(* Logix 5000 project; controller Tekno_ASRS vendor 1 type 14 code 147 rev 20.11; software revision 20.01 *)
// ASRS control program for Tekno ASRS

TASK MainTask (continuous, watchdog 500 ms) : MainProgram
TASK SafetyTask (periodic, rate 160 ms, priority 10, watchdog 20 ms) : SafetyProgram

MODULES
   Local : vendor 1 type 14 code 147 (ICP 0, rev 20.11)
      IOComms : vendor 1 type 12 code 200 (ICP 2, Ethernet 192.168.10.207, rev 5.1, Input RPI 500 ms)
         SpatulaYAxis : vendor 1 type 123 code 50 (Ethernet 192.168.10.202, rev 5.1, Output RPI 20 ms)
             : vendor 1 type 123 code 8192 (DPI 5, rev 4.1)
         XAxis : vendor 1 type 37 code 23 (Ethernet 192.168.10.200, rev 5.1, MotionDiagnostics RPI 1 ms, MotionSync RPI 6 ms)
         ZAxis : vendor 1 type 37 code 23 (Ethernet 192.168.10.201, rev 5.1, MotionDiagnostics RPI 1 ms, MotionSync RPI 6 ms)
         StationaryIO : 1734-AENT (Ethernet 192.168.10.204, rev 3.7, Output RPI 80 ms)
            StationaryIn1 : 1734-IB8 (PointIO 1, rev 3.1)
            StationaryIn3 : 1734-IB8 (PointIO 3, rev 3.1)
            StationaryIn2 : 1734-IB8 (PointIO 2, rev 3.1)
            StationaryIn4 : 1734-IB8 (PointIO 4, rev 3.1)
            StationaryStrainIn1 : vendor 1 type 0 code 20 (PointIO 5, rev 1.1, Output RPI 80 ms)
            StationarOut8 : 1734-OB8 (PointIO 8, rev 3.1)
            StationarySafetyIn1 : vendor 1 type 35 code 15 (PointIO 7, rev 1.1, Input RPI 40 ms)
            StationarySafetyOut1 : vendor 1 type 35 code 16 (PointIO 6, rev 1.1, Input RPI 320 ms, Output RPI 160 ms)
         ShuttleIO : 1734-AENT (Ethernet 192.168.10.203, rev 3.1, Output RPI 20 ms)
            ShuttleIn2 : 1734-IB8 (PointIO 2, rev 3.1)
            ShuttleIn1 : 1734-IB8 (PointIO 1, rev 3.1)
            ShuttleStrainIn1 : vendor 1 type 0 code 20 (PointIO 3, rev 1.1, Output RPI 80 ms)
            ShuttleStrainIn2 : vendor 1 type 0 code 20 (PointIO 4, rev 1.1, Output RPI 80 ms)
            ShuttleOut2 : 1734-OB8 (PointIO 10, rev 3.1)
            ShuttleOut1 : 1734-OB8 (PointIO 5, rev 3.1)
            ShuttleSafetyIn1 : vendor 1 type 35 code 15 (PointIO 7, rev 1.1, Input RPI 40 ms, Output RPI 160 ms)
            ShuttleSafetyIn2 : vendor 1 type 35 code 15 (PointIO 9, rev 1.1, Input RPI 40 ms, Output RPI 160 ms)
            ShuttleSafetyOut1 : vendor 1 type 35 code 16 (PointIO 6, rev 1.1, Input RPI 40 ms, Output RPI 160 ms)
            ShuttleSafetyOut2 : vendor 1 type 35 code 16 (PointIO 8, rev 1.1, Input RPI 40 ms, Output RPI 160 ms)
      @b5ff5b04@:Partner : vendor 1 type 14 code 146 (ICP 1, rev 20.11)   // ASRS control program for Tekno ASRS
END_MODULES

TYPE ASRS_Status :
STRUCT
   RtRowObstruction : DINT;
   LfRowObstruction : DINT;
END_STRUCT
END_TYPE

TYPE BayPos :
STRUCT
   AAxis : DINT;
   BAxis : DINT;
END_STRUCT
END_TYPE

TYPE Configuration :
STRUCT
   MaxASpeed : REAL;
   MinASpeed : REAL;
   MaxAAcc : REAL;
   MaxADec : REAL;
   AAccelJerk : REAL;
   ADecelJerk : REAL;
   MaxBSpeed : REAL;
   MinBSpeed : REAL;
   MaxBAcc : REAL;
   MaxBDec : REAL;
   BAccelJerk : REAL;
   BDecelJerk : REAL;
   SpatulaOffset : DINT;
   JogADirection : DINT;
   JogBDirection : DINT;
   AllowABSynch : BOOL;
END_STRUCT
END_TYPE

TYPE HMI_Commands :
STRUCT
   CfgEndAAxis : DINT;
   CfgEndBAxis : DINT;
   CfgStrtAAxis : DINT;
   CfgStrtBAxis : DINT;
   MaxA : DINT;
   MaxB : DINT;
   MaxC : DINT;
   GoToALocation : DINT;
   GoToBLocation : DINT;
   XLftStrainScaleSet : DINT;
   XRtStrainScaleSet : DINT;
   ZForeRtStrainScaleSet : DINT;
   ZForeLftStrainScaleSet : DINT;
   ZAftRtStrainScaleSet : DINT;
   ZAftLftStrainScaleSet : DINT;
   AGridLoc : DINT;
   BGridLoc : DINT;
   CGridLoc : DINT;
   XStrainLeftMvV : REAL;
   XStrainRightMvV : REAL;
   ZAftStrainLeftMvV : REAL;
   ZAftStrainRightMvV : REAL;
   ZForeStrainLeftMvV : REAL;
   ZForeStrainRightMvV : REAL;
   HMIStart : BOOL;
   HMIStop : BOOL;
   HMIReset : BOOL;
   JogAAxisEn : BOOL;
   JogAFwd : BOOL;
   JogARev : BOOL;
   JogBAxisEn : BOOL;
   JogBFwd : BOOL;
   JogBRev : BOOL;
   JogCAxisEn : BOOL;
   JogCFwd : BOOL;
   JogCRev : BOOL;
   ManMode : BOOL;
   ZAftRtClrTare : BOOL;
   ZAftRtTare : BOOL;
   ZAftLtClrTare : BOOL;
   ZAftLtTare : BOOL;
   ZForRTClrTare : BOOL;
   ZForRtTare : BOOL;
   ZForLtClrTare : BOOL;
   ZForLtTare : BOOL;
   XLtClrTare : BOOL;
   XLtTare : BOOL;
   XRtClrTare : BOOL;
   XRtTare : BOOL;
   SUIndPos : BOOL;
   XStCalMode : BOOL;
   XStRunMode : BOOL;
   ZAftStCalMode : BOOL;
   ZAftStRunMode : BOOL;
   ZForStCalMode : BOOL;
   ZForStRunMode : BOOL;
   GoToBay : BOOL;
   GoToHome : BOOL;
   MatrixSetUp : BOOL;
   ClearCurrent : BOOL;
   ClearQueue : BOOL;
   DemoStart : BOOL;
   DemoStop : BOOL;
   SpatulaHome : BOOL;
END_STRUCT
END_TYPE

TYPE HMI_Data :
STRUCT
   Status : HMI_Status;
   Faults : HMI_Faults;
END_STRUCT
END_TYPE

TYPE HMI_Faults :
STRUCT
   AAxisFault : DINT;
   BAxisFault : DINT;
   SystemFault : BOOL;
   AftAreaScanner : BOOL;
   EstopSafetyGate : BOOL;
   ForeAreaScanner : BOOL;
   PalmButtons : BOOL;
   RowObstruction : BOOL;
   XTension : BOOL;
   ZAftLeft : BOOL;
   ZAftRight : BOOL;
   ZForeLeft : BOOL;
   ZForeRight : BOOL;
   ShuttleFault : BOOL;
   XAxisMtrSideEOT : BOOL;
   XAxisPnlSideEOT : BOOL;
   ZAxisUpEOT : BOOL;
   ZAxisDnEOT : BOOL;
   ZLatchFault : BOOL;
   AGVLghtCurFlt : BOOL;
END_STRUCT
END_TYPE

TYPE HMI_Status :
STRUCT
   CurrentAPos : REAL;
   CurrentBPos : REAL;
   CurrentCPos : REAL;
   XStrainLeftWeight : DINT;
   XStrainRightWeight : DINT;
   ZAftStrainLeftWeight : DINT;
   ZAftStrainRightWeight : DINT;
   ZForeStrainLeftWeight : DINT;
   ZForeStrainRightWeight : DINT;
   QueuedTasks : DINT;
   AAxisStatus : DINT;
   BAxisStatus : DINT;
   CurrentTaskCommand : SINT;
   CurrentTaskBayAPos : SINT;
   CurrentTaskBayBPos : SINT;
   CurrentTaskBayCPos : SINT;
   CurrentTaskParameter1 : SINT;
   CurrentTaskParameter2 : SINT;
   Auto : BOOL;
   ManOnBoard : BOOL;
   AreaWarning : BOOL;
   ManGateClosed : BOOL;
   BackGateInstalled : BOOL;
   DrivesOn : BOOL;
   SpatulaHome : BOOL;
   SystemRunning : BOOL;
   ZLAftLft : BOOL;
   ZLAftRgt : BOOL;
   ZLForeLft : BOOL;
   ZLForeRgt : BOOL;
   FrontAreaWarn : BOOL;
   RearAreaWarn : BOOL;
   Footswitch : BOOL;
   XAxisBrk : BOOL;
   ZAxisBrk : BOOL;
   PalmButtonLeft : BOOL;
   PalmButtonright : BOOL;
END_STRUCT
END_TYPE

TYPE Messaging :
STRUCT
   Command : SINT;
   CoordinateA : SINT;
   CoordinateB : SINT;
   CoordinateC : SINT;
   Parameter1 : SINT;
   Parameter2 : SINT;
   Sequence : DINT;
END_STRUCT
END_TYPE

TYPE Position :
STRUCT
   Apos : REAL;
   Bpos : REAL;
   Cpos : REAL[10];
END_STRUCT
END_TYPE

TYPE Strain :
STRUCT
   LeftScaleSet : DINT;
   LeftAutoCalSet : DINT;
   LeftWeight : DINT;
   LeftRaw : DINT;
   LeftCal : DINT;
   RightScaleSet : DINT;
   RightAutoCalSet : DINT;
   RightWeight : DINT;
   RightRaw : DINT;
   RightCal : DINT;
   CfgAveSampCnt : DINT;
   LeftMvV : REAL;
   RightMvV : REAL;
   LeftEnAutoCal : BOOL;
   RightEnAutoCal : BOOL;
END_STRUCT
END_TYPE

TYPE Task :
STRUCT
   Command : SINT;
   BayAPos : SINT;
   BayBPos : SINT;
   BayCPos : SINT;
   Parameter1 : SINT;
   Parameter2 : SINT;
END_STRUCT
END_TYPE

VAR_GLOBAL   (* controller tags *)
   A : DINT;
   AAxis : AXIS_CIP_DRIVE;
   AAxisJog : MOTION_INSTRUCTION := (FLAGS := 33554432);
   AAxisMAM : MOTION_INSTRUCTION := (FLAGS := 167772160, PC := 1);
   AAxisMove : BOOL := 1;
   AAxisOn : MOTION_INSTRUCTION := (FLAGS := 536870912, DN := 1, STATE := 1);
   AAXisReset : MOTION_INSTRUCTION := (FLAGS := 536870912, DN := 1, STATE := 1);
   AAxisSODelay : TIMER := (PRE := 200);
   AAxisState : DINT;
   AAxisStop : MOTION_INSTRUCTION := (FLAGS := 33554432);
   ABayPos : DINT;
   ABGrid : Position[100,20] := ([0,0].Apos := 475.0, [0,0].Bpos := 0.02327277, [0,1].Apos := 63.589, [0,1].Bpos := 6.6, [0,1].Cpos[1] := -196128.0, [0,2].Apos := 677.48, [0,2].Bpos := 6.6, [0,2].Cpos[1] := -196128.0, [0,3].Apos := 46.1, [0,3].Bpos := 77.4, [0,3].Cpos[1] := -196128.0, [0,4].Apos := 80.1, [0,4].Bpos := 77.4, [0,4].Cpos[1] := -196128.0, [0,5].Apos := 660.18, [0,5].Bpos := 77.4, [0,5].Cpos[1] := -196128.0, [0,6].Apos := 694.375, [0,6].Bpos := 77.4, [0,6].Cpos[1] := -196128.0, [0,7].Apos := 415.0, [0,8].Apos := 415.0, [0,9].Apos := 415.0, [0,10].Apos := 415.0, [0,11].Apos := 415.0, [0,12].Apos := 415.0, [0,13].Apos := 415.0, [0,14].Apos := 415.0, [0,15].Apos := 415.0, [0,16].Apos := 415.0, [0,17].Apos := 415.0, [0,18].Apos := 415.0, [0,19].Apos := 415.0, [1,0].Apos := 415.0, [1,1].Apos := -42.35, [1,2].Apos := -42.35, [1,2].Bpos := 7.87817, [1,3].Apos := -42.35, [1,3].Bpos := 39.87817, [1,4].Apos := -42.35, [1,4].Bpos := 71.878174, [1,5].Apos := -42.35, [1,5].Bpos := 103.878174, [1,6].Apos := -42.35, [1,6].Bpos := 135.87817, [1,7].Apos := -42.35, [1,7].Bpos := 167.87817, [1,8].Apos := -42.35, [1,8].Bpos := 199.87817, [1,9].Apos := -42.35, [1,9].Bpos := 215.0, [1,10].Apos := 415.0, [1,11].Apos := 415.0, [1,12].Apos := 415.0, [1,13].Apos := 415.0, [1,14].Apos := 415.0, [1,15].Apos := 415.0, [1,16].Apos := 415.0, [1,17].Apos := 415.0, [1,18].Apos := 415.0,
        [1,19].Apos := 415.0, [2,0].Apos := 415.0, [2,1].Apos := -42.35, [2,2].Apos := -42.35, [2,2].Bpos := 7.87817, [2,3].Apos := -42.35, [2,3].Bpos := 39.87817, [2,4].Apos := -42.35, [2,4].Bpos := 71.878174, [2,5].Apos := -42.35, [2,5].Bpos := 103.878174, [2,6].Apos := -42.35, [2,6].Bpos := 135.87817, [2,7].Apos := -42.35, [2,7].Bpos := 167.87817, [2,8].Apos := -42.35, [2,8].Bpos := 199.87817, [2,9].Apos := -42.35, [2,9].Bpos := 215.0, [2,10].Apos := 415.0, [2,11].Apos := 415.0, [2,12].Apos := 415.0, [2,13].Apos := 415.0, [2,14].Apos := 415.0, [2,15].Apos := 415.0, [2,16].Apos := 415.0, [2,17].Apos := 415.0, [2,18].Apos := 415.0, [2,19].Apos := 415.0, [3,0].Apos := 415.0, [3,1].Apos := -26.905, [3,2].Apos := -26.905, [3,2].Bpos := 7.87817, [3,3].Apos := -26.905, [3,3].Bpos := 39.87817, [3,4].Apos := -26.905, [3,4].Bpos := 71.878174, [3,5].Apos := -26.905, [3,5].Bpos := 103.878174, [3,6].Apos := -26.905, [3,6].Bpos := 135.87817, [3,7].Apos := -26.905, [3,7].Bpos := 167.87817, [3,8].Apos := -26.905, [3,8].Bpos := 199.87817, [3,9].Apos := -26.905, [3,9].Bpos := 215.0, [3,10].Apos := 415.0, [3,11].Apos := 415.0, [3,12].Apos := 415.0, [3,13].Apos := 415.0, [3,14].Apos := 415.0, [3,15].Apos := 415.0, [3,16].Apos := 415.0, [3,17].Apos := 415.0, [3,18].Apos := 415.0, [3,19].Apos := 415.0, [4,0].Apos := 415.0, [4,1].Apos := -1.235, [4,2].Apos := -1.235,
        [4,2].Bpos := 7.87817, [4,3].Apos := -1.235, [4,3].Bpos := 39.87817, [4,4].Apos := -1.235, [4,4].Bpos := 71.878174, [4,5].Apos := -1.235, [4,5].Bpos := 103.878174, [4,6].Apos := -1.235, [4,6].Bpos := 135.87817, [4,7].Apos := -1.235, [4,7].Bpos := 167.87817, [4,8].Apos := -1.235, [4,8].Bpos := 199.87817, [4,9].Apos := -1.235, [4,9].Bpos := 215.0, [4,10].Apos := 415.0, [4,11].Apos := 415.0, [4,12].Apos := 415.0, [4,13].Apos := 415.0, [4,14].Apos := 415.0, [4,15].Apos := 415.0, [4,16].Apos := 415.0, [4,17].Apos := 415.0, [4,18].Apos := 415.0, [4,19].Apos := 415.0, [5,0].Apos := 415.0, [5,1].Apos := 24.435026, [5,2].Apos := 24.435026, [5,2].Bpos := 7.87817, [5,3].Apos := 24.435026, [5,3].Bpos := 39.87817, [5,4].Apos := 24.435026, [5,4].Bpos := 71.878174, [5,5].Apos := 24.435026, [5,5].Bpos := 103.878174, [5,6].Apos := 24.435026, [5,6].Bpos := 135.87817, [5,7].Apos := 24.435026, [5,7].Bpos := 167.87817, [5,8].Apos := 24.435026, [5,8].Bpos := 199.87817, [5,9].Apos := 24.435026, [5,9].Bpos := 215.0, [5,10].Apos := 415.0, [5,11].Apos := 415.0, [5,12].Apos := 415.0, [5,13].Apos := 415.0, [5,14].Apos := 415.0, [5,15].Apos := 415.0, [5,16].Apos := 415.0, [5,17].Apos := 415.0, [5,18].Apos := 415.0, [5,19].Apos := 415.0, [6,0].Apos := 415.0, [6,1].Apos := 50.105618, [6,2].Apos := 50.105618, [6,2].Bpos := 7.87817, [6,3].Apos := 50.105618, [6,3].Bpos := 39.87817, [6,4].Apos := 50.105618,
        [6,4].Bpos := 71.878174, [6,5].Apos := 50.105618, [6,5].Bpos := 103.878174, [6,6].Apos := 50.105618, [6,6].Bpos := 135.87817, [6,7].Apos := 50.105618, [6,7].Bpos := 167.87817, [6,8].Apos := 50.105618, [6,8].Bpos := 199.87817, [6,9].Apos := 50.105618, [6,9].Bpos := 215.0, [6,10].Apos := 415.0, [6,11].Apos := 415.0, [6,12].Apos := 415.0, [6,13].Apos := 415.0, [6,14].Apos := 415.0, [6,15].Apos := 415.0, [6,16].Apos := 415.0, [6,17].Apos := 415.0, [6,18].Apos := 415.0, [6,19].Apos := 415.0, [7,0].Apos := 415.0, [7,1].Apos := 75.77621, [7,2].Apos := 75.77621, [7,2].Bpos := 7.87817, [7,3].Apos := 75.77621, [7,3].Bpos := 39.87817, [7,4].Apos := 75.77621, [7,4].Bpos := 71.878174, [7,5].Apos := 75.77621, [7,5].Bpos := 103.878174, [7,6].Apos := 75.77621, [7,6].Bpos := 135.87817, [7,7].Apos := 75.77621, [7,7].Bpos := 167.87817, [7,8].Apos := 75.77621, [7,8].Bpos := 199.87817, [7,9].Apos := 75.77621, [7,9].Bpos := 215.0, [7,10].Apos := 415.0, [7,11].Apos := 415.0, [7,12].Apos := 415.0, [7,13].Apos := 415.0, [7,14].Apos := 415.0, [7,15].Apos := 415.0, [7,16].Apos := 415.0, [7,17].Apos := 415.0, [7,18].Apos := 415.0, [7,19].Apos := 415.0, [8,0].Apos := 415.0, [8,1].Apos := 101.4468, [8,2].Apos := 101.4468, [8,2].Bpos := 7.87817, [8,3].Apos := 101.4468, [8,3].Bpos := 39.87817, [8,4].Apos := 101.4468, [8,4].Bpos := 71.878174, [8,5].Apos := 101.4468, [8,5].Bpos := 103.878174, [8,6].Apos := 101.4468,
        [8,6].Bpos := 135.87817, [8,7].Apos := 101.4468, [8,7].Bpos := 167.87817, [8,8].Apos := 101.4468, [8,8].Bpos := 199.87817, [8,9].Apos := 101.4468, [8,9].Bpos := 215.0, [8,10].Apos := 415.0, [8,11].Apos := 415.0, [8,12].Apos := 415.0, [8,13].Apos := 415.0, [8,14].Apos := 415.0, [8,15].Apos := 415.0, [8,16].Apos := 415.0, [8,17].Apos := 415.0, [8,18].Apos := 415.0, [8,19].Apos := 415.0, [9,0].Apos := 415.0, [9,1].Apos := 127.11739, [9,2].Apos := 127.11739, [9,2].Bpos := 7.87817, [9,3].Apos := 127.11739, [9,3].Bpos := 39.87817, [9,4].Apos := 127.11739, [9,4].Bpos := 71.878174, [9,5].Apos := 127.11739, [9,5].Bpos := 103.878174, [9,6].Apos := 127.11739, [9,6].Bpos := 135.87817, [9,7].Apos := 127.11739, [9,7].Bpos := 167.87817, [9,8].Apos := 127.11739, [9,8].Bpos := 199.87817, [9,9].Apos := 127.11739, [9,9].Bpos := 215.0, [9,10].Apos := 415.0, [9,11].Apos := 415.0, [9,12].Apos := 415.0, [9,13].Apos := 415.0, [9,14].Apos := 415.0, [9,15].Apos := 415.0, [9,16].Apos := 415.0, [9,17].Apos := 415.0, [9,18].Apos := 415.0, [9,19].Apos := 415.0, [10,0].Apos := 415.0, [10,1].Apos := 152.78798, [10,2].Apos := 152.78798, [10,2].Bpos := 7.87817, [10,3].Apos := 152.78798, [10,3].Bpos := 39.87817, [10,4].Apos := 152.78798, [10,4].Bpos := 71.878174, [10,5].Apos := 152.78798, [10,5].Bpos := 103.878174, [10,6].Apos := 152.78798, [10,6].Bpos := 135.87817, [10,7].Apos := 152.78798, [10,7].Bpos := 167.87817, [10,8].Apos := 152.78798,
        [10,8].Bpos := 199.87817, [10,9].Apos := 152.78798, [10,9].Bpos := 215.0, [10,10].Apos := 415.0, [10,11].Apos := 415.0, [10,12].Apos := 415.0, [10,13].Apos := 415.0, [10,14].Apos := 415.0, [10,15].Apos := 415.0, [10,16].Apos := 415.0, [10,17].Apos := 415.0, [10,18].Apos := 415.0, [10,19].Apos := 415.0, [11,0].Apos := 415.0, [11,1].Apos := 178.45857, [11,2].Apos := 178.45857, [11,2].Bpos := 7.87817, [11,3].Apos := 178.45857, [11,3].Bpos := 39.87817, [11,4].Apos := 178.45857, [11,4].Bpos := 71.878174, [11,5].Apos := 178.45857, [11,5].Bpos := 103.878174, [11,6].Apos := 178.45857, [11,6].Bpos := 135.87817, [11,7].Apos := 178.45857, [11,7].Bpos := 167.87817, [11,8].Apos := 178.45857, [11,8].Bpos := 199.87817, [11,9].Apos := 178.45857, [11,9].Bpos := 215.0, [11,10].Apos := 415.0, [11,11].Apos := 415.0, [11,12].Apos := 415.0, [11,13].Apos := 415.0, [11,14].Apos := 415.0, [11,15].Apos := 415.0, [11,16].Apos := 415.0, [11,17].Apos := 415.0, [11,18].Apos := 415.0, [11,19].Apos := 415.0, [12,0].Apos := 415.0, [12,1].Apos := 204.12917, [12,2].Apos := 204.12917, [12,2].Bpos := 7.87817, [12,3].Apos := 204.12917, [12,3].Bpos := 39.87817, [12,4].Apos := 204.12917, [12,4].Bpos := 71.878174, [12,5].Apos := 204.12917, [12,5].Bpos := 103.878174, [12,6].Apos := 204.12917, [12,6].Bpos := 135.87817, [12,7].Apos := 204.12917, [12,7].Bpos := 167.87817, [12,8].Apos := 204.12917, [12,8].Bpos := 199.87817, [12,9].Apos := 204.12917, [12,9].Bpos := 215.0, [12,10].Apos := 415.0,
        [12,11].Apos := 415.0, [12,12].Apos := 415.0, [12,13].Apos := 415.0, [12,14].Apos := 415.0, [12,15].Apos := 415.0, [12,16].Apos := 415.0, [12,17].Apos := 415.0, [12,18].Apos := 415.0, [12,19].Apos := 415.0, [13,0].Apos := 415.0, [13,1].Apos := 229.79976, [13,2].Apos := 229.79976, [13,2].Bpos := 7.87817, [13,3].Apos := 229.79976, [13,3].Bpos := 39.87817, [13,4].Apos := 229.79976, [13,4].Bpos := 71.878174, [13,5].Apos := 229.79976, [13,5].Bpos := 103.878174, [13,6].Apos := 229.79976, [13,6].Bpos := 135.87817, [13,7].Apos := 229.79976, [13,7].Bpos := 167.87817, [13,8].Apos := 229.79976, [13,8].Bpos := 199.87817, [13,9].Apos := 229.79976, [13,9].Bpos := 215.0, [13,10].Apos := 415.0, [13,11].Apos := 415.0, [13,12].Apos := 415.0, [13,13].Apos := 415.0, [13,14].Apos := 415.0, [13,15].Apos := 415.0, [13,16].Apos := 415.0, [13,17].Apos := 415.0, [13,18].Apos := 415.0, [13,19].Apos := 415.0, [14,0].Apos := 415.0, [14,1].Apos := 255.47035, [14,2].Apos := 255.47035, [14,2].Bpos := 7.87817, [14,3].Apos := 255.47035, [14,3].Bpos := 39.87817, [14,4].Apos := 255.47035, [14,4].Bpos := 71.878174, [14,5].Apos := 255.47035, [14,5].Bpos := 103.878174, [14,6].Apos := 255.47035, [14,6].Bpos := 135.87817, [14,7].Apos := 255.47035, [14,7].Bpos := 167.87817, [14,8].Apos := 255.47035, [14,8].Bpos := 199.87817, [14,9].Apos := 255.47035, [14,9].Bpos := 215.0, [14,10].Apos := 415.0, [14,11].Apos := 415.0, [14,12].Apos := 415.0, [14,13].Apos := 415.0, [14,14].Apos := 415.0,
        [14,15].Apos := 415.0, [14,16].Apos := 415.0, [14,17].Apos := 415.0, [14,18].Apos := 415.0, [14,19].Apos := 415.0, [15,0].Apos := 415.0, [15,1].Apos := 281.14093, [15,2].Apos := 281.14093, [15,2].Bpos := 7.87817, [15,3].Apos := 281.14093, [15,3].Bpos := 39.87817, [15,4].Apos := 281.14093, [15,4].Bpos := 71.878174, [15,5].Apos := 281.14093, [15,5].Bpos := 103.878174, [15,6].Apos := 281.14093, [15,6].Bpos := 135.87817, [15,7].Apos := 281.14093, [15,7].Bpos := 167.87817, [15,8].Apos := 281.14093, [15,8].Bpos := 199.87817, [15,9].Apos := 281.14093, [15,9].Bpos := 215.0, [15,10].Apos := 415.0, [15,11].Apos := 415.0, [15,12].Apos := 415.0, [15,13].Apos := 415.0, [15,14].Apos := 415.0, [15,15].Apos := 415.0, [15,16].Apos := 415.0, [15,17].Apos := 415.0, [15,18].Apos := 415.0, [15,19].Apos := 415.0, [16,0].Apos := 415.0, [16,1].Apos := 306.81152, [16,2].Apos := 306.81152, [16,2].Bpos := 7.87817, [16,3].Apos := 306.81152, [16,3].Bpos := 39.87817, [16,4].Apos := 306.81152, [16,4].Bpos := 71.878174, [16,5].Apos := 306.81152, [16,5].Bpos := 103.878174, [16,6].Apos := 306.81152, [16,6].Bpos := 135.87817, [16,7].Apos := 306.81152, [16,7].Bpos := 167.87817, [16,8].Apos := 306.81152, [16,8].Bpos := 199.87817, [16,9].Apos := 306.81152, [16,9].Bpos := 215.0, [16,10].Apos := 415.0, [16,11].Apos := 415.0, [16,12].Apos := 415.0, [16,13].Apos := 415.0, [16,14].Apos := 415.0, [16,15].Apos := 415.0, [16,16].Apos := 415.0, [16,17].Apos := 415.0, [16,18].Apos := 415.0,
        [16,19].Apos := 415.0, [17,0].Apos := 415.0, [17,1].Apos := 332.48212, [17,2].Apos := 332.48212, [17,2].Bpos := 7.87817, [17,3].Apos := 332.48212, [17,3].Bpos := 39.87817, [17,4].Apos := 332.48212, [17,4].Bpos := 71.878174, [17,5].Apos := 332.48212, [17,5].Bpos := 103.878174, [17,6].Apos := 332.48212, [17,6].Bpos := 135.87817, [17,7].Apos := 332.48212, [17,7].Bpos := 167.87817, [17,8].Apos := 332.48212, [17,8].Bpos := 199.87817, [17,9].Apos := 332.48212, [17,9].Bpos := 215.0, [17,10].Apos := 415.0, [17,11].Apos := 415.0, [17,12].Apos := 415.0, [17,13].Apos := 415.0, [17,14].Apos := 415.0, [17,15].Apos := 415.0, [17,16].Apos := 415.0, [17,17].Apos := 415.0, [17,18].Apos := 415.0, [17,19].Apos := 415.0, [18,0].Apos := 415.0, [18,1].Apos := 358.1527, [18,2].Apos := 358.1527, [18,2].Bpos := 7.87817, [18,3].Apos := 358.1527, [18,3].Bpos := 39.87817, [18,4].Apos := 358.1527, [18,4].Bpos := 71.878174, [18,5].Apos := 358.1527, [18,5].Bpos := 103.878174, [18,6].Apos := 358.1527, [18,6].Bpos := 135.87817, [18,7].Apos := 358.1527, [18,7].Bpos := 167.87817, [18,8].Apos := 358.1527, [18,8].Bpos := 199.87817, [18,9].Apos := 358.1527, [18,9].Bpos := 215.0, [18,10].Apos := 415.0, [18,11].Apos := 415.0, [18,12].Apos := 415.0, [18,13].Apos := 415.0, [18,14].Apos := 415.0, [18,15].Apos := 415.0, [18,16].Apos := 415.0, [18,17].Apos := 415.0, [18,18].Apos := 415.0, [18,19].Apos := 415.0, [19,0].Apos := 415.0, [19,1].Apos := 383.8233, [19,2].Apos := 383.8233,
        [19,2].Bpos := 7.87817, [19,3].Apos := 383.8233, [19,3].Bpos := 39.87817, [19,4].Apos := 383.8233, [19,4].Bpos := 71.878174, [19,5].Apos := 383.8233, [19,5].Bpos := 103.878174, [19,6].Apos := 383.8233, [19,6].Bpos := 135.87817, [19,7].Apos := 383.8233, [19,7].Bpos := 167.87817, [19,8].Apos := 383.8233, [19,8].Bpos := 199.87817, [19,9].Apos := 383.8233, [19,9].Bpos := 215.0, [19,10].Apos := 415.0, [19,11].Apos := 415.0, [19,12].Apos := 415.0, [19,13].Apos := 415.0, [19,14].Apos := 415.0, [19,15].Apos := 415.0, [19,16].Apos := 415.0, [19,17].Apos := 415.0, [19,18].Apos := 415.0, [19,19].Apos := 415.0, [20,0].Apos := 415.0, [20,1].Apos := 409.4939, [20,2].Apos := 409.4939, [20,2].Bpos := 7.87817, [20,3].Apos := 409.4939, [20,3].Bpos := 39.87817, [20,4].Apos := 409.4939, [20,4].Bpos := 71.878174, [20,5].Apos := 409.4939, [20,5].Bpos := 103.878174, [20,6].Apos := 409.4939, [20,6].Bpos := 135.87817, [20,7].Apos := 409.4939, [20,7].Bpos := 167.87817, [20,8].Apos := 409.4939, [20,8].Bpos := 199.87817, [20,9].Apos := 409.4939, [20,9].Bpos := 215.0, [20,10].Apos := 415.0, [20,11].Apos := 415.0, [20,12].Apos := 415.0, [20,13].Apos := 415.0, [20,14].Apos := 415.0, [20,15].Apos := 415.0, [20,16].Apos := 415.0, [20,17].Apos := 415.0, [20,18].Apos := 415.0, [20,19].Apos := 415.0, [21,0].Apos := 415.0, [21,1].Apos := 435.1645, [21,2].Apos := 435.1645, [21,2].Bpos := 7.87817, [21,3].Apos := 435.1645, [21,3].Bpos := 39.87817, [21,4].Apos := 435.1645,
        [21,4].Bpos := 71.878174, [21,5].Apos := 435.1645, [21,5].Bpos := 103.878174, [21,6].Apos := 435.1645, [21,6].Bpos := 135.87817, [21,7].Apos := 435.1645, [21,7].Bpos := 167.87817, [21,8].Apos := 435.1645, [21,8].Bpos := 199.87817, [21,9].Apos := 435.1645, [21,9].Bpos := 215.0, [21,10].Apos := 415.0, [21,11].Apos := 415.0, [21,12].Apos := 415.0, [21,13].Apos := 415.0, [21,14].Apos := 415.0, [21,15].Apos := 415.0, [21,16].Apos := 415.0, [21,17].Apos := 415.0, [21,18].Apos := 415.0, [21,19].Apos := 415.0, [22,0].Apos := 415.0, [22,1].Apos := 460.83508, [22,2].Apos := 460.83508, [22,2].Bpos := 7.87817, [22,3].Apos := 460.83508, [22,3].Bpos := 39.87817, [22,4].Apos := 460.83508, [22,4].Bpos := 71.878174, [22,5].Apos := 460.83508, [22,5].Bpos := 103.878174, [22,6].Apos := 460.83508, [22,6].Bpos := 135.87817, [22,7].Apos := 460.83508, [22,7].Bpos := 167.87817, [22,8].Apos := 460.83508, [22,8].Bpos := 199.87817, [22,9].Apos := 460.83508, [22,9].Bpos := 215.0, [22,10].Apos := 415.0, [22,11].Apos := 415.0, [22,12].Apos := 415.0, [22,13].Apos := 415.0, [22,14].Apos := 415.0, [22,15].Apos := 415.0, [22,16].Apos := 415.0, [22,17].Apos := 415.0, [22,18].Apos := 415.0, [22,19].Apos := 415.0, [23,0].Apos := 415.0, [23,1].Apos := 486.50568, [23,2].Apos := 486.50568, [23,2].Bpos := 7.87817, [23,3].Apos := 486.50568, [23,3].Bpos := 39.87817, [23,4].Apos := 486.50568, [23,4].Bpos := 71.878174, [23,5].Apos := 486.50568, [23,5].Bpos := 103.878174, [23,6].Apos := 486.50568,
        [23,6].Bpos := 135.87817, [23,7].Apos := 486.50568, [23,7].Bpos := 167.87817, [23,8].Apos := 486.50568, [23,8].Bpos := 199.87817, [23,9].Apos := 486.50568, [23,9].Bpos := 215.0, [23,10].Apos := 415.0, [23,11].Apos := 415.0, [23,12].Apos := 415.0, [23,13].Apos := 415.0, [23,14].Apos := 415.0, [23,15].Apos := 415.0, [23,16].Apos := 415.0, [23,17].Apos := 415.0, [23,18].Apos := 415.0, [23,19].Apos := 415.0, [24,0].Apos := 415.0, [24,1].Apos := 512.1763, [24,2].Apos := 512.1763, [24,2].Bpos := 7.87817, [24,3].Apos := 512.1763, [24,3].Bpos := 39.87817, [24,4].Apos := 512.1763, [24,4].Bpos := 71.878174, [24,5].Apos := 512.1763, [24,5].Bpos := 103.878174, [24,6].Apos := 512.1763, [24,6].Bpos := 135.87817, [24,7].Apos := 512.1763, [24,7].Bpos := 167.87817, [24,8].Apos := 512.1763, [24,8].Bpos := 199.87817, [24,9].Apos := 512.1763, [24,9].Bpos := 215.0, [24,10].Apos := 415.0, [24,11].Apos := 415.0, [24,12].Apos := 415.0, [24,13].Apos := 415.0, [24,14].Apos := 415.0, [24,15].Apos := 415.0, [24,16].Apos := 415.0, [24,17].Apos := 415.0, [24,18].Apos := 415.0, [24,19].Apos := 415.0, [25,0].Apos := 415.0, [25,1].Apos := 537.8468, [25,2].Apos := 537.8468, [25,2].Bpos := 7.87817, [25,3].Apos := 537.8468, [25,3].Bpos := 39.87817, [25,4].Apos := 537.8468, [25,4].Bpos := 71.878174, [25,5].Apos := 537.8468, [25,5].Bpos := 103.878174, [25,6].Apos := 537.8468, [25,6].Bpos := 135.87817, [25,7].Apos := 537.8468, [25,7].Bpos := 167.87817, [25,8].Apos := 537.8468,
        [25,8].Bpos := 199.87817, [25,9].Apos := 537.8468, [25,9].Bpos := 215.0, [25,10].Apos := 415.0, [25,11].Apos := 415.0, [25,12].Apos := 415.0, [25,13].Apos := 415.0, [25,14].Apos := 415.0, [25,15].Apos := 415.0, [25,16].Apos := 415.0, [25,17].Apos := 415.0, [25,18].Apos := 415.0, [25,19].Apos := 415.0, [26,0].Apos := 415.0, [26,1].Apos := 563.5174, [26,2].Apos := 563.5174, [26,2].Bpos := 7.87817, [26,3].Apos := 563.5174, [26,3].Bpos := 39.87817, [26,4].Apos := 563.5174, [26,4].Bpos := 71.878174, [26,5].Apos := 563.5174, [26,5].Bpos := 103.878174, [26,6].Apos := 563.5174, [26,6].Bpos := 135.87817, [26,7].Apos := 563.5174, [26,7].Bpos := 167.87817, [26,8].Apos := 563.5174, [26,8].Bpos := 199.87817, [26,9].Apos := 563.5174, [26,9].Bpos := 215.0, [26,10].Apos := 415.0, [26,11].Apos := 415.0, [26,12].Apos := 415.0, [26,13].Apos := 415.0, [26,14].Apos := 415.0, [26,15].Apos := 415.0, [26,16].Apos := 415.0, [26,17].Apos := 415.0, [26,18].Apos := 415.0, [26,19].Apos := 415.0, [27,0].Apos := 415.0, [27,1].Apos := 589.188, [27,2].Apos := 589.188, [27,2].Bpos := 7.87817, [27,3].Apos := 589.188, [27,3].Bpos := 39.87817, [27,4].Apos := 589.188, [27,4].Bpos := 71.878174, [27,5].Apos := 589.188, [27,5].Bpos := 103.878174, [27,6].Apos := 589.188, [27,6].Bpos := 135.87817, [27,7].Apos := 589.188, [27,7].Bpos := 167.87817, [27,8].Apos := 589.188, [27,8].Bpos := 199.87817, [27,9].Apos := 589.188, [27,9].Bpos := 215.0, [27,10].Apos := 415.0,
        [27,11].Apos := 415.0, [27,12].Apos := 415.0, [27,13].Apos := 415.0, [27,14].Apos := 415.0, [27,15].Apos := 415.0, [27,16].Apos := 415.0, [27,17].Apos := 415.0, [27,18].Apos := 415.0, [27,19].Apos := 415.0, [28,0].Apos := 415.0, [28,1].Apos := 614.8586, [28,2].Apos := 614.8586, [28,2].Bpos := 7.87817, [28,3].Apos := 614.8586, [28,3].Bpos := 39.87817, [28,4].Apos := 614.8586, [28,4].Bpos := 71.878174, [28,5].Apos := 614.8586, [28,5].Bpos := 103.878174, [28,6].Apos := 614.8586, [28,6].Bpos := 135.87817, [28,7].Apos := 614.8586, [28,7].Bpos := 167.87817, [28,8].Apos := 614.8586, [28,8].Bpos := 199.87817, [28,9].Apos := 614.8586, [28,9].Bpos := 215.0, [28,10].Apos := 415.0, [28,11].Apos := 415.0, [28,12].Apos := 415.0, [28,13].Apos := 415.0, [28,14].Apos := 415.0, [28,15].Apos := 415.0, [28,16].Apos := 415.0, [28,17].Apos := 415.0, [28,18].Apos := 415.0, [28,19].Apos := 415.0, [29,0].Apos := 415.0, [29,1].Apos := 640.5292, [29,2].Apos := 640.5292, [29,2].Bpos := 7.87817, [29,3].Apos := 640.5292, [29,3].Bpos := 39.87817, [29,4].Apos := 640.5292, [29,4].Bpos := 71.878174, [29,5].Apos := 640.5292, [29,5].Bpos := 103.878174, [29,6].Apos := 640.5292, [29,6].Bpos := 135.87817, [29,7].Apos := 640.5292, [29,7].Bpos := 167.87817, [29,8].Apos := 640.5292, [29,8].Bpos := 199.87817, [29,9].Apos := 640.5292, [29,9].Bpos := 215.0, [29,10].Apos := 415.0, [29,11].Apos := 415.0, [29,12].Apos := 415.0, [29,13].Apos := 415.0, [29,14].Apos := 415.0,
        [29,15].Apos := 415.0, [29,16].Apos := 415.0, [29,17].Apos := 415.0, [29,18].Apos := 415.0, [29,19].Apos := 415.0, [30,0].Apos := 415.0, [30,1].Apos := 666.19977, [30,2].Apos := 666.19977, [30,2].Bpos := 7.87817, [30,3].Apos := 666.19977, [30,3].Bpos := 39.87817, [30,4].Apos := 666.19977, [30,4].Bpos := 71.878174, [30,5].Apos := 666.19977, [30,5].Bpos := 103.878174, [30,6].Apos := 666.19977, [30,6].Bpos := 135.87817, [30,7].Apos := 666.19977, [30,7].Bpos := 167.87817, [30,8].Apos := 666.19977, [30,8].Bpos := 199.87817, [30,9].Apos := 666.19977, [30,9].Bpos := 215.0, [30,10].Apos := 415.0, [30,11].Apos := 415.0, [30,12].Apos := 415.0, [30,13].Apos := 415.0, [30,14].Apos := 415.0, [30,15].Apos := 415.0, [30,16].Apos := 415.0, [30,17].Apos := 415.0, [30,18].Apos := 415.0, [30,19].Apos := 415.0, [31,0].Apos := 415.0, [31,1].Apos := 691.87036, [31,2].Apos := 691.87036, [31,2].Bpos := 7.87817, [31,3].Apos := 691.87036, [31,3].Bpos := 39.87817, [31,4].Apos := 691.87036, [31,4].Bpos := 71.878174, [31,5].Apos := 691.87036, [31,5].Bpos := 103.878174, [31,6].Apos := 691.87036, [31,6].Bpos := 135.87817, [31,7].Apos := 691.87036, [31,7].Bpos := 167.87817, [31,8].Apos := 691.87036, [31,8].Bpos := 199.87817, [31,9].Apos := 691.87036, [31,9].Bpos := 215.0, [31,10].Apos := 415.0, [31,11].Apos := 415.0, [31,12].Apos := 415.0, [31,13].Apos := 415.0, [31,14].Apos := 415.0, [31,15].Apos := 415.0, [31,16].Apos := 415.0, [31,17].Apos := 415.0, [31,18].Apos := 415.0,
        [31,19].Apos := 415.0, [32,0].Apos := 415.0, [32,1].Apos := 717.54095, [32,2].Apos := 717.54095, [32,2].Bpos := 7.87817, [32,3].Apos := 717.54095, [32,3].Bpos := 39.87817, [32,4].Apos := 717.54095, [32,4].Bpos := 71.878174, [32,5].Apos := 717.54095, [32,5].Bpos := 103.878174, [32,6].Apos := 717.54095, [32,6].Bpos := 135.87817, [32,7].Apos := 717.54095, [32,7].Bpos := 167.87817, [32,8].Apos := 717.54095, [32,8].Bpos := 199.87817, [32,9].Apos := 717.54095, [32,9].Bpos := 215.0, [32,10].Apos := 415.0, [32,11].Apos := 415.0, [32,12].Apos := 415.0, [32,13].Apos := 415.0, [32,14].Apos := 415.0, [32,15].Apos := 415.0, [32,16].Apos := 415.0, [32,17].Apos := 415.0, [32,18].Apos := 415.0, [32,19].Apos := 415.0, [33,0].Apos := 415.0, [33,1].Apos := 743.21155, [33,2].Apos := 743.21155, [33,2].Bpos := 7.87817, [33,3].Apos := 743.21155, [33,3].Bpos := 39.87817, [33,4].Apos := 743.21155, [33,4].Bpos := 71.878174, [33,5].Apos := 743.21155, [33,5].Bpos := 103.878174, [33,6].Apos := 743.21155, [33,6].Bpos := 135.87817, [33,7].Apos := 743.21155, [33,7].Bpos := 167.87817, [33,8].Apos := 743.21155, [33,8].Bpos := 199.87817, [33,9].Apos := 743.21155, [33,9].Bpos := 215.0, [33,10].Apos := 415.0, [33,11].Apos := 415.0, [33,12].Apos := 415.0, [33,13].Apos := 415.0, [33,14].Apos := 415.0, [33,15].Apos := 415.0, [33,16].Apos := 415.0, [33,17].Apos := 415.0, [33,18].Apos := 415.0, [33,19].Apos := 415.0, [34,0].Apos := 415.0, [34,1].Apos := 768.88214, [34,2].Apos := 768.88214,
        [34,2].Bpos := 7.87817, [34,3].Apos := 768.88214, [34,3].Bpos := 39.87817, [34,4].Apos := 768.88214, [34,4].Bpos := 71.878174, [34,5].Apos := 768.88214, [34,5].Bpos := 103.878174, [34,6].Apos := 768.88214, [34,6].Bpos := 135.87817, [34,7].Apos := 768.88214, [34,7].Bpos := 167.87817, [34,8].Apos := 768.88214, [34,8].Bpos := 199.87817, [34,9].Apos := 768.88214, [34,9].Bpos := 215.0, [34,10].Apos := 415.0, [34,11].Apos := 415.0, [34,12].Apos := 415.0, [34,13].Apos := 415.0, [34,14].Apos := 415.0, [34,15].Apos := 415.0, [34,16].Apos := 415.0, [34,17].Apos := 415.0, [34,18].Apos := 415.0, [34,19].Apos := 415.0, [35,0].Apos := 415.0, [35,1].Apos := 794.55273, [35,2].Apos := 794.55273, [35,2].Bpos := 7.87817, [35,3].Apos := 794.55273, [35,3].Bpos := 39.87817, [35,4].Apos := 794.55273, [35,4].Bpos := 71.878174, [35,5].Apos := 794.55273, [35,5].Bpos := 103.878174, [35,6].Apos := 794.55273, [35,6].Bpos := 135.87817, [35,7].Apos := 794.55273, [35,7].Bpos := 167.87817, [35,8].Apos := 794.55273, [35,8].Bpos := 199.87817, [35,9].Apos := 794.55273, [35,9].Bpos := 215.0, [35,10].Apos := 415.0, [35,11].Apos := 415.0, [35,12].Apos := 415.0, [35,13].Apos := 415.0, [35,14].Apos := 415.0, [35,15].Apos := 415.0, [35,16].Apos := 415.0, [35,17].Apos := 415.0, [35,18].Apos := 415.0, [35,19].Apos := 415.0, [36,0].Apos := 415.0, [36,1].Apos := 820.2233, [36,2].Apos := 820.2233, [36,2].Bpos := 7.87817, [36,3].Apos := 820.2233, [36,3].Bpos := 39.87817, [36,4].Apos := 820.2233,
        [36,4].Bpos := 71.878174, [36,5].Apos := 820.2233, [36,5].Bpos := 103.878174, [36,6].Apos := 820.2233, [36,6].Bpos := 135.87817, [36,7].Apos := 820.2233, [36,7].Bpos := 167.87817, [36,8].Apos := 820.2233, [36,8].Bpos := 199.87817, [36,9].Apos := 820.2233, [36,9].Bpos := 215.0, [36,10].Apos := 415.0, [36,11].Apos := 415.0, [36,12].Apos := 415.0, [36,13].Apos := 415.0, [36,14].Apos := 415.0, [36,15].Apos := 415.0, [36,16].Apos := 415.0, [36,17].Apos := 415.0, [36,18].Apos := 415.0, [36,19].Apos := 415.0, [37,0].Apos := 415.0, [37,1].Apos := 845.89, [37,2].Apos := 845.89, [37,2].Bpos := 8.0, [37,3].Apos := 845.89, [37,3].Bpos := 40.0, [37,4].Apos := 845.89, [37,4].Bpos := 72.0, [37,5].Apos := 845.89, [37,5].Bpos := 104.0, [37,6].Apos := 845.89, [37,6].Bpos := 136.0, [37,7].Apos := 845.89, [37,7].Bpos := 168.0, [37,8].Apos := 845.89, [37,8].Bpos := 200.0, [37,9].Apos := 845.89, [37,9].Bpos := 215.0, [37,10].Apos := 415.0, [37,11].Apos := 415.0, [37,12].Apos := 415.0, [37,13].Apos := 415.0, [37,14].Apos := 415.0, [37,15].Apos := 415.0, [37,16].Apos := 415.0, [37,17].Apos := 415.0, [37,18].Apos := 415.0, [37,19].Apos := 415.0, [38,0].Apos := 415.0, [38,1].Apos := 871.6, [38,2].Apos := 871.6, [38,2].Bpos := 8.0, [38,3].Apos := 871.6, [38,3].Bpos := 40.0, [38,4].Apos := 871.6, [38,4].Bpos := 72.0, [38,5].Apos := 871.6, [38,5].Bpos := 104.0, [38,6].Apos := 871.6,
        [38,6].Bpos := 136.0, [38,7].Apos := 871.6, [38,7].Bpos := 168.0, [38,8].Apos := 871.6, [38,8].Bpos := 200.0, [38,9].Apos := 871.6, [38,9].Bpos := 215.0, [38,10].Apos := 415.0, [38,11].Apos := 415.0, [38,12].Apos := 415.0, [38,13].Apos := 415.0, [38,14].Apos := 415.0, [38,15].Apos := 415.0, [38,16].Apos := 415.0, [38,17].Apos := 415.0, [38,18].Apos := 415.0, [38,19].Apos := 415.0, [39,0].Apos := 415.0, [39,1].Apos := 887.0, [39,2].Apos := 887.0, [39,2].Bpos := 8.0, [39,3].Apos := 887.0, [39,3].Bpos := 40.0, [39,4].Apos := 887.0, [39,4].Bpos := 72.0, [39,5].Apos := 887.0, [39,5].Bpos := 104.0, [39,6].Apos := 887.0, [39,6].Bpos := 136.0, [39,7].Apos := 887.0, [39,7].Bpos := 168.0, [39,8].Apos := 887.0, [39,8].Bpos := 200.0, [39,9].Apos := 887.0, [39,9].Bpos := 215.0, [39,10].Apos := 415.0, [39,11].Apos := 415.0, [39,12].Apos := 415.0, [39,13].Apos := 415.0, [39,14].Apos := 415.0, [39,15].Apos := 415.0, [39,16].Apos := 415.0, [39,17].Apos := 415.0, [39,18].Apos := 415.0, [39,19].Apos := 415.0, [40,0].Apos := 415.0, [40,1].Apos := 887.0, [40,2].Apos := 887.0, [40,2].Bpos := 8.0, [40,3].Apos := 887.0, [40,3].Bpos := 40.0, [40,4].Apos := 887.0, [40,4].Bpos := 72.0, [40,5].Apos := 887.0, [40,5].Bpos := 104.0, [40,6].Apos := 887.0, [40,6].Bpos := 136.0, [40,7].Apos := 887.0, [40,7].Bpos := 168.0, [40,8].Apos := 887.0,
        [40,8].Bpos := 200.0, [40,9].Apos := 887.0, [40,9].Bpos := 215.0, [40,10].Apos := 415.0, [40,11].Apos := 415.0, [40,12].Apos := 415.0, [40,13].Apos := 415.0, [40,14].Apos := 415.0, [40,15].Apos := 415.0, [40,16].Apos := 415.0, [40,17].Apos := 415.0, [40,18].Apos := 415.0, [40,19].Apos := 415.0, [41,0].Apos := 415.0, [41,1].Apos := 415.0, [41,2].Apos := 415.0, [41,3].Apos := 415.0, [41,4].Apos := 415.0, [41,5].Apos := 415.0, [41,6].Apos := 415.0, [41,7].Apos := 415.0, [41,8].Apos := 415.0, [41,9].Apos := 415.0, [41,10].Apos := 415.0, [41,11].Apos := 415.0, [41,12].Apos := 415.0, [41,13].Apos := 415.0, [41,14].Apos := 415.0, [41,15].Apos := 415.0, [41,16].Apos := 415.0, [41,17].Apos := 415.0, [41,18].Apos := 415.0, [41,19].Apos := 415.0, [42,0].Apos := 415.0, [42,1].Apos := 415.0, [42,2].Apos := 415.0, [42,3].Apos := 415.0, [42,4].Apos := 415.0, [42,5].Apos := 415.0, [42,6].Apos := 415.0, [42,7].Apos := 415.0, [42,8].Apos := 415.0, [42,9].Apos := 415.0, [42,10].Apos := 415.0, [42,11].Apos := 415.0, [42,12].Apos := 415.0, [42,13].Apos := 415.0, [42,14].Apos := 415.0, [42,15].Apos := 415.0, [42,16].Apos := 415.0, [42,17].Apos := 415.0, [42,18].Apos := 415.0, [42,19].Apos := 415.0, [43,0].Apos := 415.0, [43,1].Apos := 415.0, [43,2].Apos := 415.0, [43,3].Apos := 415.0, [43,4].Apos := 415.0, [43,5].Apos := 415.0, [43,6].Apos := 415.0,
        [43,7].Apos := 415.0, [43,8].Apos := 415.0, [43,9].Apos := 415.0, [43,10].Apos := 415.0, [43,11].Apos := 415.0, [43,12].Apos := 415.0, [43,13].Apos := 415.0, [43,14].Apos := 415.0, [43,15].Apos := 415.0, [43,16].Apos := 415.0, [43,17].Apos := 415.0, [43,18].Apos := 415.0, [43,19].Apos := 415.0, [44,0].Apos := 415.0, [44,1].Apos := 415.0, [44,2].Apos := 415.0, [44,3].Apos := 415.0, [44,4].Apos := 415.0, [44,5].Apos := 415.0, [44,6].Apos := 415.0, [44,7].Apos := 415.0, [44,8].Apos := 415.0, [44,9].Apos := 415.0, [44,10].Apos := 415.0, [44,11].Apos := 415.0, [44,12].Apos := 415.0, [44,13].Apos := 415.0, [44,14].Apos := 415.0, [44,15].Apos := 415.0, [44,16].Apos := 415.0, [44,17].Apos := 415.0, [44,18].Apos := 415.0, [44,19].Apos := 415.0, [45,0].Apos := 415.0, [45,1].Apos := 415.0, [45,2].Apos := 415.0, [45,3].Apos := 415.0, [45,4].Apos := 415.0, [45,5].Apos := 415.0, [45,6].Apos := 415.0, [45,7].Apos := 415.0, [45,8].Apos := 415.0, [45,9].Apos := 415.0, [45,10].Apos := 415.0, [45,11].Apos := 415.0, [45,12].Apos := 415.0, [45,13].Apos := 415.0, [45,14].Apos := 415.0, [45,15].Apos := 415.0, [45,16].Apos := 415.0, [45,17].Apos := 415.0, [45,18].Apos := 415.0, [45,19].Apos := 415.0, [46,0].Apos := 415.0, [46,1].Apos := 415.0, [46,2].Apos := 415.0, [46,3].Apos := 415.0, [46,4].Apos := 415.0, [46,5].Apos := 415.0, [46,6].Apos := 415.0,
        [46,7].Apos := 415.0, [46,8].Apos := 415.0, [46,9].Apos := 415.0, [46,10].Apos := 415.0, [46,11].Apos := 415.0, [46,12].Apos := 415.0, [46,13].Apos := 415.0, [46,14].Apos := 415.0, [46,15].Apos := 415.0, [46,16].Apos := 415.0, [46,17].Apos := 415.0, [46,18].Apos := 415.0, [46,19].Apos := 415.0, [47,0].Apos := 415.0, [47,1].Apos := 415.0, [47,2].Apos := 415.0, [47,3].Apos := 415.0, [47,4].Apos := 415.0, [47,5].Apos := 415.0, [47,6].Apos := 415.0, [47,7].Apos := 415.0, [47,8].Apos := 415.0, [47,9].Apos := 415.0, [47,10].Apos := 415.0, [47,11].Apos := 415.0, [47,12].Apos := 415.0, [47,13].Apos := 415.0, [47,14].Apos := 415.0, [47,15].Apos := 415.0, [47,16].Apos := 415.0, [47,17].Apos := 415.0, [47,18].Apos := 415.0, [47,19].Apos := 415.0, [48,0].Apos := 415.0, [48,1].Apos := 415.0, [48,2].Apos := 415.0, [48,3].Apos := 415.0, [48,4].Apos := 415.0, [48,5].Apos := 415.0, [48,6].Apos := 415.0, [48,7].Apos := 415.0, [48,8].Apos := 415.0, [48,9].Apos := 415.0, [48,10].Apos := 415.0, [48,11].Apos := 415.0, [48,12].Apos := 415.0, [48,13].Apos := 415.0, [48,14].Apos := 415.0, [48,15].Apos := 415.0, [48,16].Apos := 415.0, [48,17].Apos := 415.0, [48,18].Apos := 415.0, [48,19].Apos := 415.0, [49,0].Apos := 415.0, [49,1].Apos := 415.0, [49,2].Apos := 415.0, [49,3].Apos := 415.0, [49,4].Apos := 415.0, [49,5].Apos := 415.0, [49,6].Apos := 415.0,
        [49,7].Apos := 415.0, [49,8].Apos := 415.0, [49,9].Apos := 415.0, [49,10].Apos := 415.0, [49,11].Apos := 415.0, [49,12].Apos := 415.0, [49,13].Apos := 415.0, [49,14].Apos := 415.0, [49,15].Apos := 415.0, [49,16].Apos := 415.0, [49,17].Apos := 415.0, [49,18].Apos := 415.0, [49,19].Apos := 415.0, [50,0].Apos := 415.0, [50,1].Apos := 415.0, [50,2].Apos := 415.0, [50,3].Apos := 415.0, [50,4].Apos := 415.0, [50,5].Apos := 415.0, [50,6].Apos := 415.0, [50,7].Apos := 415.0, [50,8].Apos := 415.0, [50,9].Apos := 415.0, [50,10].Apos := 415.0, [50,11].Apos := 415.0, [50,12].Apos := 415.0, [50,13].Apos := 415.0, [50,14].Apos := 415.0, [50,15].Apos := 415.0, [50,16].Apos := 415.0, [50,17].Apos := 415.0, [50,18].Apos := 415.0, [50,19].Apos := 415.0, [51,0].Apos := 415.0, [51,1].Apos := 415.0, [51,2].Apos := 415.0, [51,3].Apos := 415.0, [51,4].Apos := 415.0, [51,5].Apos := 415.0, [51,6].Apos := 415.0, [51,7].Apos := 415.0, [51,8].Apos := 415.0, [51,9].Apos := 415.0, [51,10].Apos := 415.0, [51,11].Apos := 415.0, [51,12].Apos := 415.0, [51,13].Apos := 415.0, [51,14].Apos := 415.0, [51,15].Apos := 415.0, [51,16].Apos := 415.0, [51,17].Apos := 415.0, [51,18].Apos := 415.0, [51,19].Apos := 415.0, [52,0].Apos := 415.0, [52,1].Apos := 415.0, [52,2].Apos := 415.0, [52,3].Apos := 415.0, [52,4].Apos := 415.0, [52,5].Apos := 415.0, [52,6].Apos := 415.0,
        [52,7].Apos := 415.0, [52,8].Apos := 415.0, [52,9].Apos := 415.0, [52,10].Apos := 415.0, [52,11].Apos := 415.0, [52,12].Apos := 415.0, [52,13].Apos := 415.0, [52,14].Apos := 415.0, [52,15].Apos := 415.0, [52,16].Apos := 415.0, [52,17].Apos := 415.0, [52,18].Apos := 415.0, [52,19].Apos := 415.0, [53,0].Apos := 415.0, [53,1].Apos := 415.0, [53,2].Apos := 415.0, [53,3].Apos := 415.0, [53,4].Apos := 415.0, [53,5].Apos := 415.0, [53,6].Apos := 415.0, [53,7].Apos := 415.0, [53,8].Apos := 415.0, [53,9].Apos := 415.0, [53,10].Apos := 415.0, [53,11].Apos := 415.0, [53,12].Apos := 415.0, [53,13].Apos := 415.0, [53,14].Apos := 415.0, [53,15].Apos := 415.0, [53,16].Apos := 415.0, [53,17].Apos := 415.0, [53,18].Apos := 415.0, [53,19].Apos := 415.0, [54,0].Apos := 415.0, [54,1].Apos := 415.0, [54,2].Apos := 415.0, [54,3].Apos := 415.0, [54,4].Apos := 415.0, [54,5].Apos := 415.0, [54,6].Apos := 415.0, [54,7].Apos := 415.0, [54,8].Apos := 415.0, [54,9].Apos := 415.0, [54,10].Apos := 415.0, [54,11].Apos := 415.0, [54,12].Apos := 415.0, [54,13].Apos := 415.0, [54,14].Apos := 415.0, [54,15].Apos := 415.0, [54,16].Apos := 415.0, [54,17].Apos := 415.0, [54,18].Apos := 415.0, [54,19].Apos := 415.0, [55,0].Apos := 415.0, [55,1].Apos := 415.0, [55,2].Apos := 415.0, [55,3].Apos := 415.0, [55,4].Apos := 415.0, [55,5].Apos := 415.0, [55,6].Apos := 415.0,
        [55,7].Apos := 415.0, [55,8].Apos := 415.0, [55,9].Apos := 415.0, [55,10].Apos := 415.0, [55,11].Apos := 415.0, [55,12].Apos := 415.0, [55,13].Apos := 415.0, [55,14].Apos := 415.0, [55,15].Apos := 415.0, [55,16].Apos := 415.0, [55,17].Apos := 415.0, [55,18].Apos := 415.0, [55,19].Apos := 415.0, [56,0].Apos := 415.0, [56,1].Apos := 415.0, [56,2].Apos := 415.0, [56,3].Apos := 415.0, [56,4].Apos := 415.0, [56,5].Apos := 415.0, [56,6].Apos := 415.0, [56,7].Apos := 415.0, [56,8].Apos := 415.0, [56,9].Apos := 415.0, [56,10].Apos := 415.0, [56,11].Apos := 415.0, [56,12].Apos := 415.0, [56,13].Apos := 415.0, [56,14].Apos := 415.0, [56,15].Apos := 415.0, [56,16].Apos := 415.0, [56,17].Apos := 415.0, [56,18].Apos := 415.0, [56,19].Apos := 415.0, [57,0].Apos := 415.0, [57,1].Apos := 415.0, [57,2].Apos := 415.0, [57,3].Apos := 415.0, [57,4].Apos := 415.0, [57,5].Apos := 415.0, [57,6].Apos := 415.0, [57,7].Apos := 415.0, [57,8].Apos := 415.0, [57,9].Apos := 415.0, [57,10].Apos := 415.0, [57,11].Apos := 415.0, [57,12].Apos := 415.0, [57,13].Apos := 415.0, [57,14].Apos := 415.0, [57,15].Apos := 415.0, [57,16].Apos := 415.0, [57,17].Apos := 415.0, [57,18].Apos := 415.0, [57,19].Apos := 415.0, [58,0].Apos := 415.0, [58,1].Apos := 415.0, [58,2].Apos := 415.0, [58,3].Apos := 415.0, [58,4].Apos := 415.0, [58,5].Apos := 415.0, [58,6].Apos := 415.0,
        [58,7].Apos := 415.0, [58,8].Apos := 415.0, [58,9].Apos := 415.0, [58,10].Apos := 415.0, [58,11].Apos := 415.0, [58,12].Apos := 415.0, [58,13].Apos := 415.0, [58,14].Apos := 415.0, [58,15].Apos := 415.0, [58,16].Apos := 415.0, [58,17].Apos := 415.0, [58,18].Apos := 415.0, [58,19].Apos := 415.0, [59,0].Apos := 415.0, [59,1].Apos := 415.0, [59,2].Apos := 415.0, [59,3].Apos := 415.0, [59,4].Apos := 415.0, [59,5].Apos := 415.0, [59,6].Apos := 415.0, [59,7].Apos := 415.0, [59,8].Apos := 415.0, [59,9].Apos := 415.0, [59,10].Apos := 415.0, [59,11].Apos := 415.0, [59,12].Apos := 415.0, [59,13].Apos := 415.0, [59,14].Apos := 415.0, [59,15].Apos := 415.0, [59,16].Apos := 415.0, [59,17].Apos := 415.0, [59,18].Apos := 415.0, [59,19].Apos := 415.0, [60,0].Apos := 415.0, [60,1].Apos := 415.0, [60,2].Apos := 415.0, [60,3].Apos := 415.0, [60,4].Apos := 415.0, [60,5].Apos := 415.0, [60,6].Apos := 415.0, [60,7].Apos := 415.0, [60,8].Apos := 415.0, [60,9].Apos := 415.0, [60,10].Apos := 415.0, [60,11].Apos := 415.0, [60,12].Apos := 415.0, [60,13].Apos := 415.0, [60,14].Apos := 415.0, [60,15].Apos := 415.0, [60,16].Apos := 415.0, [60,17].Apos := 415.0, [60,18].Apos := 415.0, [60,19].Apos := 415.0, [61,0].Apos := 415.0, [61,1].Apos := 415.0, [61,2].Apos := 415.0, [61,3].Apos := 415.0, [61,4].Apos := 415.0, [61,5].Apos := 415.0, [61,6].Apos := 415.0,
        [61,7].Apos := 415.0, [61,8].Apos := 415.0, [61,9].Apos := 415.0, [61,10].Apos := 415.0, [61,11].Apos := 415.0, [61,12].Apos := 415.0, [61,13].Apos := 415.0, [61,14].Apos := 415.0, [61,15].Apos := 415.0, [61,16].Apos := 415.0, [61,17].Apos := 415.0, [61,18].Apos := 415.0, [61,19].Apos := 415.0, [62,0].Apos := 415.0, [62,1].Apos := 415.0, [62,2].Apos := 415.0, [62,3].Apos := 415.0, [62,4].Apos := 415.0, [62,5].Apos := 415.0, [62,6].Apos := 415.0, [62,7].Apos := 415.0, [62,8].Apos := 415.0, [62,9].Apos := 415.0, [62,10].Apos := 415.0, [62,11].Apos := 415.0, [62,12].Apos := 415.0, [62,13].Apos := 415.0, [62,14].Apos := 415.0, [62,15].Apos := 415.0, [62,16].Apos := 415.0, [62,17].Apos := 415.0, [62,18].Apos := 415.0, [62,19].Apos := 415.0, [63,0].Apos := 415.0, [63,1].Apos := 415.0, [63,2].Apos := 415.0, [63,3].Apos := 415.0, [63,4].Apos := 415.0, [63,5].Apos := 415.0, [63,6].Apos := 415.0, [63,7].Apos := 415.0, [63,8].Apos := 415.0, [63,9].Apos := 415.0, [63,10].Apos := 415.0, [63,11].Apos := 415.0, [63,12].Apos := 415.0, [63,13].Apos := 415.0, [63,14].Apos := 415.0, [63,15].Apos := 415.0, [63,16].Apos := 415.0, [63,17].Apos := 415.0, [63,18].Apos := 415.0, [63,19].Apos := 415.0, [64,0].Apos := 415.0, [64,1].Apos := 415.0, [64,2].Apos := 415.0, [64,3].Apos := 415.0, [64,4].Apos := 415.0, [64,5].Apos := 415.0, [64,6].Apos := 415.0,
        [64,7].Apos := 415.0, [64,8].Apos := 415.0, [64,9].Apos := 415.0, [64,10].Apos := 415.0, [64,11].Apos := 415.0, [64,12].Apos := 415.0, [64,13].Apos := 415.0, [64,14].Apos := 415.0, [64,15].Apos := 415.0, [64,16].Apos := 415.0, [64,17].Apos := 415.0, [64,18].Apos := 415.0, [64,19].Apos := 415.0, [65,0].Apos := 415.0, [65,1].Apos := 415.0, [65,2].Apos := 415.0, [65,3].Apos := 415.0, [65,4].Apos := 415.0, [65,5].Apos := 415.0, [65,6].Apos := 415.0, [65,7].Apos := 415.0, [65,8].Apos := 415.0, [65,9].Apos := 415.0, [65,10].Apos := 415.0, [65,11].Apos := 415.0, [65,12].Apos := 415.0, [65,13].Apos := 415.0, [65,14].Apos := 415.0, [65,15].Apos := 415.0, [65,16].Apos := 415.0, [65,17].Apos := 415.0, [65,18].Apos := 415.0, [65,19].Apos := 415.0, [66,0].Apos := 415.0, [66,1].Apos := 415.0, [66,2].Apos := 415.0, [66,3].Apos := 415.0, [66,4].Apos := 415.0, [66,5].Apos := 415.0, [66,6].Apos := 415.0, [66,7].Apos := 415.0, [66,8].Apos := 415.0, [66,9].Apos := 415.0, [66,10].Apos := 415.0, [66,11].Apos := 415.0, [66,12].Apos := 415.0, [66,13].Apos := 415.0, [66,14].Apos := 415.0, [66,15].Apos := 415.0, [66,16].Apos := 415.0, [66,17].Apos := 415.0, [66,18].Apos := 415.0, [66,19].Apos := 415.0, [67,0].Apos := 415.0, [67,1].Apos := 415.0, [67,2].Apos := 415.0, [67,3].Apos := 415.0, [67,4].Apos := 415.0, [67,5].Apos := 415.0, [67,6].Apos := 415.0,
        [67,7].Apos := 415.0, [67,8].Apos := 415.0, [67,9].Apos := 415.0, [67,10].Apos := 415.0, [67,11].Apos := 415.0, [67,12].Apos := 415.0, [67,13].Apos := 415.0, [67,14].Apos := 415.0, [67,15].Apos := 415.0, [67,16].Apos := 415.0, [67,17].Apos := 415.0, [67,18].Apos := 415.0, [67,19].Apos := 415.0, [68,0].Apos := 415.0, [68,1].Apos := 415.0, [68,2].Apos := 415.0, [68,3].Apos := 415.0, [68,4].Apos := 415.0, [68,5].Apos := 415.0, [68,6].Apos := 415.0, [68,7].Apos := 415.0, [68,8].Apos := 415.0, [68,9].Apos := 415.0, [68,10].Apos := 415.0, [68,11].Apos := 415.0, [68,12].Apos := 415.0, [68,13].Apos := 415.0, [68,14].Apos := 415.0, [68,15].Apos := 415.0, [68,16].Apos := 415.0, [68,17].Apos := 415.0, [68,18].Apos := 415.0, [68,19].Apos := 415.0, [69,0].Apos := 415.0, [69,1].Apos := 415.0, [69,2].Apos := 415.0, [69,3].Apos := 415.0, [69,4].Apos := 415.0, [69,5].Apos := 415.0, [69,6].Apos := 415.0, [69,7].Apos := 415.0, [69,8].Apos := 415.0, [69,9].Apos := 415.0, [69,10].Apos := 415.0, [69,11].Apos := 415.0, [69,12].Apos := 415.0, [69,13].Apos := 415.0, [69,14].Apos := 415.0, [69,15].Apos := 415.0, [69,16].Apos := 415.0, [69,17].Apos := 415.0, [69,18].Apos := 415.0, [69,19].Apos := 415.0, [70,0].Apos := 415.0, [70,1].Apos := 415.0, [70,2].Apos := 415.0, [70,3].Apos := 415.0, [70,4].Apos := 415.0, [70,5].Apos := 415.0, [70,6].Apos := 415.0,
        [70,7].Apos := 415.0, [70,8].Apos := 415.0, [70,9].Apos := 415.0, [70,10].Apos := 415.0, [70,11].Apos := 415.0, [70,12].Apos := 415.0, [70,13].Apos := 415.0, [70,14].Apos := 415.0, [70,15].Apos := 415.0, [70,16].Apos := 415.0, [70,17].Apos := 415.0, [70,18].Apos := 415.0, [70,19].Apos := 415.0, [71,0].Apos := 415.0, [71,1].Apos := 415.0, [71,2].Apos := 415.0, [71,3].Apos := 415.0, [71,4].Apos := 415.0, [71,5].Apos := 415.0, [71,6].Apos := 415.0, [71,7].Apos := 415.0, [71,8].Apos := 415.0, [71,9].Apos := 415.0, [71,10].Apos := 415.0, [71,11].Apos := 415.0, [71,12].Apos := 415.0, [71,13].Apos := 415.0, [71,14].Apos := 415.0, [71,15].Apos := 415.0, [71,16].Apos := 415.0, [71,17].Apos := 415.0, [71,18].Apos := 415.0, [71,19].Apos := 415.0, [72,0].Apos := 415.0, [72,1].Apos := 415.0, [72,2].Apos := 415.0, [72,3].Apos := 415.0, [72,4].Apos := 415.0, [72,5].Apos := 415.0, [72,6].Apos := 415.0, [72,7].Apos := 415.0, [72,8].Apos := 415.0, [72,9].Apos := 415.0, [72,10].Apos := 415.0, [72,11].Apos := 415.0, [72,12].Apos := 415.0, [72,13].Apos := 415.0, [72,14].Apos := 415.0, [72,15].Apos := 415.0, [72,16].Apos := 415.0, [72,17].Apos := 415.0, [72,18].Apos := 415.0, [72,19].Apos := 415.0, [73,0].Apos := 415.0, [73,1].Apos := 415.0, [73,2].Apos := 415.0, [73,3].Apos := 415.0, [73,4].Apos := 415.0, [73,5].Apos := 415.0, [73,6].Apos := 415.0,
        [73,7].Apos := 415.0, [73,8].Apos := 415.0, [73,9].Apos := 415.0, [73,10].Apos := 415.0, [73,11].Apos := 415.0, [73,12].Apos := 415.0, [73,13].Apos := 415.0, [73,14].Apos := 415.0, [73,15].Apos := 415.0, [73,16].Apos := 415.0, [73,17].Apos := 415.0, [73,18].Apos := 415.0, [73,19].Apos := 415.0, [74,0].Apos := 415.0, [74,1].Apos := 415.0, [74,2].Apos := 415.0, [74,3].Apos := 415.0, [74,4].Apos := 415.0, [74,5].Apos := 415.0, [74,6].Apos := 415.0, [74,7].Apos := 415.0, [74,8].Apos := 415.0, [74,9].Apos := 415.0, [74,10].Apos := 415.0, [74,11].Apos := 415.0, [74,12].Apos := 415.0, [74,13].Apos := 415.0, [74,14].Apos := 415.0, [74,15].Apos := 415.0, [74,16].Apos := 415.0, [74,17].Apos := 415.0, [74,18].Apos := 415.0, [74,19].Apos := 415.0, [75,0].Apos := 415.0, [75,1].Apos := 415.0, [75,2].Apos := 415.0, [75,3].Apos := 415.0, [75,4].Apos := 415.0, [75,5].Apos := 415.0, [75,6].Apos := 415.0, [75,7].Apos := 415.0, [75,8].Apos := 415.0, [75,9].Apos := 415.0, [75,10].Apos := 415.0, [75,11].Apos := 415.0, [75,12].Apos := 415.0, [75,13].Apos := 415.0, [75,14].Apos := 415.0, [75,15].Apos := 415.0, [75,16].Apos := 415.0, [75,17].Apos := 415.0, [75,18].Apos := 415.0, [75,19].Apos := 415.0, [76,0].Apos := 415.0, [76,1].Apos := 415.0, [76,2].Apos := 415.0, [76,3].Apos := 415.0, [76,4].Apos := 415.0, [76,5].Apos := 415.0, [76,6].Apos := 415.0,
        [76,7].Apos := 415.0, [76,8].Apos := 415.0, [76,9].Apos := 415.0, [76,10].Apos := 415.0, [76,11].Apos := 415.0, [76,12].Apos := 415.0, [76,13].Apos := 415.0, [76,14].Apos := 415.0, [76,15].Apos := 415.0, [76,16].Apos := 415.0, [76,17].Apos := 415.0, [76,18].Apos := 415.0, [76,19].Apos := 415.0, [77,0].Apos := 415.0, [77,1].Apos := 415.0, [77,2].Apos := 415.0, [77,3].Apos := 415.0, [77,4].Apos := 415.0, [77,5].Apos := 415.0, [77,6].Apos := 415.0, [77,7].Apos := 415.0, [77,8].Apos := 415.0, [77,9].Apos := 415.0, [77,10].Apos := 415.0, [77,11].Apos := 415.0, [77,12].Apos := 415.0, [77,13].Apos := 415.0, [77,14].Apos := 415.0, [77,15].Apos := 415.0, [77,16].Apos := 415.0, [77,17].Apos := 415.0, [77,18].Apos := 415.0, [77,19].Apos := 415.0, [78,0].Apos := 415.0, [78,1].Apos := 415.0, [78,2].Apos := 415.0, [78,3].Apos := 415.0, [78,4].Apos := 415.0, [78,5].Apos := 415.0, [78,6].Apos := 415.0, [78,7].Apos := 415.0, [78,8].Apos := 415.0, [78,9].Apos := 415.0, [78,10].Apos := 415.0, [78,11].Apos := 415.0, [78,12].Apos := 415.0, [78,13].Apos := 415.0, [78,14].Apos := 415.0, [78,15].Apos := 415.0, [78,16].Apos := 415.0, [78,17].Apos := 415.0, [78,18].Apos := 415.0, [78,19].Apos := 415.0, [79,0].Apos := 415.0, [79,1].Apos := 415.0, [79,2].Apos := 415.0, [79,3].Apos := 415.0, [79,4].Apos := 415.0, [79,5].Apos := 415.0, [79,6].Apos := 415.0,
        [79,7].Apos := 415.0, [79,8].Apos := 415.0, [79,9].Apos := 415.0, [79,10].Apos := 415.0, [79,11].Apos := 415.0, [79,12].Apos := 415.0, [79,13].Apos := 415.0, [79,14].Apos := 415.0, [79,15].Apos := 415.0, [79,16].Apos := 415.0, [79,17].Apos := 415.0, [79,18].Apos := 415.0, [79,19].Apos := 415.0, [80,0].Apos := 415.0, [80,1].Apos := 415.0, [80,2].Apos := 415.0, [80,3].Apos := 415.0, [80,4].Apos := 415.0, [80,5].Apos := 415.0, [80,6].Apos := 415.0, [80,7].Apos := 415.0, [80,8].Apos := 415.0, [80,9].Apos := 415.0, [80,10].Apos := 415.0, [80,11].Apos := 415.0, [80,12].Apos := 415.0, [80,13].Apos := 415.0, [80,14].Apos := 415.0, [80,15].Apos := 415.0, [80,16].Apos := 415.0, [80,17].Apos := 415.0, [80,18].Apos := 415.0, [80,19].Apos := 415.0, [81,0].Apos := 415.0, [81,1].Apos := 415.0, [81,2].Apos := 415.0, [81,3].Apos := 415.0, [81,4].Apos := 415.0, [81,5].Apos := 415.0, [81,6].Apos := 415.0, [81,7].Apos := 415.0, [81,8].Apos := 415.0, [81,9].Apos := 415.0, [81,10].Apos := 415.0, [81,11].Apos := 415.0, [81,12].Apos := 415.0, [81,13].Apos := 415.0, [81,14].Apos := 415.0, [81,15].Apos := 415.0, [81,16].Apos := 415.0, [81,17].Apos := 415.0, [81,18].Apos := 415.0, [81,19].Apos := 415.0, [82,0].Apos := 415.0, [82,1].Apos := 415.0, [82,2].Apos := 415.0, [82,3].Apos := 415.0, [82,4].Apos := 415.0, [82,5].Apos := 415.0, [82,6].Apos := 415.0,
        [82,7].Apos := 415.0, [82,8].Apos := 415.0, [82,9].Apos := 415.0, [82,10].Apos := 415.0, [82,11].Apos := 415.0, [82,12].Apos := 415.0, [82,13].Apos := 415.0, [82,14].Apos := 415.0, [82,15].Apos := 415.0, [82,16].Apos := 415.0, [82,17].Apos := 415.0, [82,18].Apos := 415.0, [82,19].Apos := 415.0, [83,0].Apos := 415.0, [83,1].Apos := 415.0, [83,2].Apos := 415.0, [83,3].Apos := 415.0, [83,4].Apos := 415.0, [83,5].Apos := 415.0, [83,6].Apos := 415.0, [83,7].Apos := 415.0, [83,8].Apos := 415.0, [83,9].Apos := 415.0, [83,10].Apos := 415.0, [83,11].Apos := 415.0, [83,12].Apos := 415.0, [83,13].Apos := 415.0, [83,14].Apos := 415.0, [83,15].Apos := 415.0, [83,16].Apos := 415.0, [83,17].Apos := 415.0, [83,18].Apos := 415.0, [83,19].Apos := 415.0, [84,0].Apos := 415.0, [84,1].Apos := 415.0, [84,2].Apos := 415.0, [84,3].Apos := 415.0, [84,4].Apos := 415.0, [84,5].Apos := 415.0, [84,6].Apos := 415.0, [84,7].Apos := 415.0, [84,8].Apos := 415.0, [84,9].Apos := 415.0, [84,10].Apos := 415.0, [84,11].Apos := 415.0, [84,12].Apos := 415.0, [84,13].Apos := 415.0, [84,14].Apos := 415.0, [84,15].Apos := 415.0, [84,16].Apos := 415.0, [84,17].Apos := 415.0, [84,18].Apos := 415.0, [84,19].Apos := 415.0, [85,0].Apos := 415.0, [85,1].Apos := 415.0, [85,2].Apos := 415.0, [85,3].Apos := 415.0, [85,4].Apos := 415.0, [85,5].Apos := 415.0, [85,6].Apos := 415.0,
        [85,7].Apos := 415.0, [85,8].Apos := 415.0, [85,9].Apos := 415.0, [85,10].Apos := 415.0, [85,11].Apos := 415.0, [85,12].Apos := 415.0, [85,13].Apos := 415.0, [85,14].Apos := 415.0, [85,15].Apos := 415.0, [85,16].Apos := 415.0, [85,17].Apos := 415.0, [85,18].Apos := 415.0, [85,19].Apos := 415.0, [86,0].Apos := 415.0, [86,1].Apos := 415.0, [86,2].Apos := 415.0, [86,3].Apos := 415.0, [86,4].Apos := 415.0, [86,5].Apos := 415.0, [86,6].Apos := 415.0, [86,7].Apos := 415.0, [86,8].Apos := 415.0, [86,9].Apos := 415.0, [86,10].Apos := 415.0, [86,11].Apos := 415.0, [86,12].Apos := 415.0, [86,13].Apos := 415.0, [86,14].Apos := 415.0, [86,15].Apos := 415.0, [86,16].Apos := 415.0, [86,17].Apos := 415.0, [86,18].Apos := 415.0, [86,19].Apos := 415.0, [87,0].Apos := 415.0, [87,1].Apos := 415.0, [87,2].Apos := 415.0, [87,3].Apos := 415.0, [87,4].Apos := 415.0, [87,5].Apos := 415.0, [87,6].Apos := 415.0, [87,7].Apos := 415.0, [87,8].Apos := 415.0, [87,9].Apos := 415.0, [87,10].Apos := 415.0, [87,11].Apos := 415.0, [87,12].Apos := 415.0, [87,13].Apos := 415.0, [87,14].Apos := 415.0, [87,15].Apos := 415.0, [87,16].Apos := 415.0, [87,17].Apos := 415.0, [87,18].Apos := 415.0, [87,19].Apos := 415.0, [88,0].Apos := 415.0, [88,1].Apos := 415.0, [88,2].Apos := 415.0, [88,3].Apos := 415.0, [88,4].Apos := 415.0, [88,5].Apos := 415.0, [88,6].Apos := 415.0,
        [88,7].Apos := 415.0, [88,8].Apos := 415.0, [88,9].Apos := 415.0, [88,10].Apos := 415.0, [88,11].Apos := 415.0, [88,12].Apos := 415.0, [88,13].Apos := 415.0, [88,14].Apos := 415.0, [88,15].Apos := 415.0, [88,16].Apos := 415.0, [88,17].Apos := 415.0, [88,18].Apos := 415.0, [88,19].Apos := 415.0, [89,0].Apos := 415.0, [89,1].Apos := 415.0, [89,2].Apos := 415.0, [89,3].Apos := 415.0, [89,4].Apos := 415.0, [89,5].Apos := 415.0, [89,6].Apos := 415.0, [89,7].Apos := 415.0, [89,8].Apos := 415.0, [89,9].Apos := 415.0, [89,10].Apos := 415.0, [89,11].Apos := 415.0, [89,12].Apos := 415.0, [89,13].Apos := 415.0, [89,14].Apos := 415.0, [89,15].Apos := 415.0, [89,16].Apos := 415.0, [89,17].Apos := 415.0, [89,18].Apos := 415.0, [89,19].Apos := 415.0, [90,0].Apos := 415.0, [90,1].Apos := 415.0, [90,2].Apos := 415.0, [90,3].Apos := 415.0, [90,4].Apos := 415.0, [90,5].Apos := 415.0, [90,6].Apos := 415.0, [90,7].Apos := 415.0, [90,8].Apos := 415.0, [90,9].Apos := 415.0, [90,10].Apos := 415.0, [90,11].Apos := 415.0, [90,12].Apos := 415.0, [90,13].Apos := 415.0, [90,14].Apos := 415.0, [90,15].Apos := 415.0, [90,16].Apos := 415.0, [90,17].Apos := 415.0, [90,18].Apos := 415.0, [90,19].Apos := 415.0, [91,0].Apos := 415.0, [91,1].Apos := 415.0, [91,2].Apos := 415.0, [91,3].Apos := 415.0, [91,4].Apos := 415.0, [91,5].Apos := 415.0, [91,6].Apos := 415.0,
        [91,7].Apos := 415.0, [91,8].Apos := 415.0, [91,9].Apos := 415.0, [91,10].Apos := 415.0, [91,11].Apos := 415.0, [91,12].Apos := 415.0, [91,13].Apos := 415.0, [91,14].Apos := 415.0, [91,15].Apos := 415.0, [91,16].Apos := 415.0, [91,17].Apos := 415.0, [91,18].Apos := 415.0, [91,19].Apos := 415.0, [92,0].Apos := 415.0, [92,1].Apos := 415.0, [92,2].Apos := 415.0, [92,3].Apos := 415.0, [92,4].Apos := 415.0, [92,5].Apos := 415.0, [92,6].Apos := 415.0, [92,7].Apos := 415.0, [92,8].Apos := 415.0, [92,9].Apos := 415.0, [92,10].Apos := 415.0, [92,11].Apos := 415.0, [92,12].Apos := 415.0, [92,13].Apos := 415.0, [92,14].Apos := 415.0, [92,15].Apos := 415.0, [92,16].Apos := 415.0, [92,17].Apos := 415.0, [92,18].Apos := 415.0, [92,19].Apos := 415.0, [93,0].Apos := 415.0, [93,1].Apos := 415.0, [93,2].Apos := 415.0, [93,3].Apos := 415.0, [93,4].Apos := 415.0, [93,5].Apos := 415.0, [93,6].Apos := 415.0, [93,7].Apos := 415.0, [93,8].Apos := 415.0, [93,9].Apos := 415.0, [93,10].Apos := 415.0, [93,11].Apos := 415.0, [93,12].Apos := 415.0, [93,13].Apos := 415.0, [93,14].Apos := 415.0, [93,15].Apos := 415.0, [93,16].Apos := 415.0, [93,17].Apos := 415.0, [93,18].Apos := 415.0, [93,19].Apos := 415.0, [94,0].Apos := 415.0, [94,1].Apos := 415.0, [94,2].Apos := 415.0, [94,3].Apos := 415.0, [94,4].Apos := 415.0, [94,5].Apos := 415.0, [94,6].Apos := 415.0,
        [94,7].Apos := 415.0, [94,8].Apos := 415.0, [94,9].Apos := 415.0, [94,10].Apos := 415.0, [94,11].Apos := 415.0, [94,12].Apos := 415.0, [94,13].Apos := 415.0, [94,14].Apos := 415.0, [94,15].Apos := 415.0, [94,16].Apos := 415.0, [94,17].Apos := 415.0, [94,18].Apos := 415.0, [94,19].Apos := 415.0, [95,0].Apos := 415.0, [95,1].Apos := 415.0, [95,2].Apos := 415.0, [95,3].Apos := 415.0, [95,4].Apos := 415.0, [95,5].Apos := 415.0, [95,6].Apos := 415.0, [95,7].Apos := 415.0, [95,8].Apos := 415.0, [95,9].Apos := 415.0, [95,10].Apos := 415.0, [95,11].Apos := 415.0, [95,12].Apos := 415.0, [95,13].Apos := 415.0, [95,14].Apos := 415.0, [95,15].Apos := 415.0, [95,16].Apos := 415.0, [95,17].Apos := 415.0, [95,18].Apos := 415.0, [95,19].Apos := 415.0, [96,0].Apos := 415.0, [96,1].Apos := 415.0, [96,2].Apos := 415.0, [96,3].Apos := 415.0, [96,4].Apos := 415.0, [96,5].Apos := 415.0, [96,6].Apos := 415.0, [96,7].Apos := 415.0, [96,8].Apos := 415.0, [96,9].Apos := 415.0, [96,10].Apos := 415.0, [96,11].Apos := 415.0, [96,12].Apos := 415.0, [96,13].Apos := 415.0, [96,14].Apos := 415.0, [96,15].Apos := 415.0, [96,16].Apos := 415.0, [96,17].Apos := 415.0, [96,18].Apos := 415.0, [96,19].Apos := 415.0, [97,0].Apos := 415.0, [97,1].Apos := 415.0, [97,2].Apos := 415.0, [97,3].Apos := 415.0, [97,4].Apos := 415.0, [97,5].Apos := 415.0, [97,6].Apos := 415.0,
        [97,7].Apos := 415.0, [97,8].Apos := 415.0, [97,9].Apos := 415.0, [97,10].Apos := 415.0, [97,11].Apos := 415.0, [97,12].Apos := 415.0, [97,13].Apos := 415.0, [97,14].Apos := 415.0, [97,15].Apos := 415.0, [97,16].Apos := 415.0, [97,17].Apos := 415.0, [97,18].Apos := 415.0, [97,19].Apos := 415.0, [98,0].Apos := 415.0, [98,1].Apos := 415.0, [98,2].Apos := 415.0, [98,3].Apos := 415.0, [98,4].Apos := 415.0, [98,5].Apos := 415.0, [98,6].Apos := 415.0, [98,7].Apos := 415.0, [98,8].Apos := 415.0, [98,9].Apos := 415.0, [98,10].Apos := 415.0, [98,11].Apos := 415.0, [98,12].Apos := 415.0, [98,13].Apos := 415.0, [98,14].Apos := 415.0, [98,15].Apos := 415.0, [98,16].Apos := 415.0, [98,17].Apos := 415.0, [98,18].Apos := 415.0, [98,19].Apos := 415.0, [99,0].Apos := 415.0, [99,1].Apos := 415.0, [99,2].Apos := 415.0, [99,3].Apos := 415.0, [99,4].Apos := 415.0, [99,5].Apos := 415.0, [99,6].Apos := 415.0, [99,7].Apos := 415.0, [99,8].Apos := 415.0, [99,9].Apos := 415.0, [99,10].Apos := 415.0, [99,11].Apos := 415.0, [99,12].Apos := 415.0, [99,13].Apos := 415.0, [99,14].Apos := 415.0, [99,15].Apos := 415.0, [99,16].Apos := 415.0, [99,17].Apos := 415.0, [99,18].Apos := 415.0, [99,19].Apos := 415.0);
   ACompare : REAL := 24.435026;
   ACoordSetup : BOOL;
   advalue : DINT := 1;
   advalue2 : DINT := 3;
   AEnableONS : BOOL := 1;
   AEnd : DINT := 15;
   AftAreaRest : ALIAS FOR ShuttleIO:8:O.Pt05Data;
   AftAreaRst : ALIAS FOR ShuttleIO:8:O.Pt04Data;
   AftAreaScanner : DCI_STOP := (ChannelA := 1, ChannelB := 1, InputStatus := 1, RestartType := 1, ColdStartType := 1, SafetyFunction := 3, DiscrepancyTime := 500, O1 := 1);
   AftAreaZn1 : ALIAS FOR ShuttleIO:8:O.Pt07Data;
   AftAreaZn2 : ALIAS FOR ShuttleIO:10:O.2;
   AftAreaZn4 : ALIAS FOR ShuttleIO:8:O.Pt06Data;
   AftEndZn : BOOL := 1;
   AftEndZnLimit : DINT := 55;
   AftEndZone : BOOL := 1;
   AgridLoc : DINT;
   AGVatDP : ALIAS FOR StationaryIO:1:I.3;
   AGVatPU : ALIAS FOR StationaryIO:1:I.2;
   AGVDP : BOOL;
   AGVLightCurtains : DCI_STOP := (InputStatus := 1, RestartType := 1, ColdStartType := 1, SafetyFunction := 2, DiscrepancyTime := 300);
   AGVok2LvDP : ALIAS FOR StationaryIO:8:O.0;
   AGVok2LvPU : ALIAS FOR StationaryIO:8:O.1;
   AGVPU : BOOL;
   AGVPUHoldTmr : TIMER := (PRE := 10000);
   AInc : DINT;
   AisleClear : BOOL := 1;
   AllowSynchAB : BOOL := 1;
   APitch : REAL;
   APos : REAL := 415.0;
   ARange : REAL;
   AreaToggle : BOOL;
   AreaWarn : ALIAS FOR ShuttleIO:5:O.2;
   AReq : DINT := 5;
   AReqPos : REAL := 24.435026;
   ASRSEnable : BOOL;
   ASRSMCR : BOOL;
   ASRSStatus : ASRS_Status;
   AStart : REAL := 415.0;
   AutoConfig : Configuration := (MaxASpeed := 150.0, MaxAAcc := 40.0, MaxADec := 40.0, AAccelJerk := 40.0, ADecelJerk := 40.0, MaxBSpeed := 50.0, MaxBAcc := 20.0, MaxBDec := 20.0, BAccelJerk := 40.0, BDecelJerk := 40.0, SpatulaOffset := 6);
   AutoMode : BOOL;
   AxisEnabled : BOOL;
   AxisStateMask : DINT := 2817;
   AxisStateReady : BOOL := 1;
   B : DINT;
   BackGateInstalled : ALIAS FOR ShuttleIO:9:I.Pt01Data;
   BAxis : AXIS_CIP_DRIVE;
   BAxisJog : MOTION_INSTRUCTION := (FLAGS := 33554432);
   BAxisMAM : MOTION_INSTRUCTION := (FLAGS := 167772160, PC := 1);
   BAxisMove : BOOL;
   BAxisOn : MOTION_INSTRUCTION := (FLAGS := 536870912, DN := 1, STATE := 1);
   BAXisReset : MOTION_INSTRUCTION := (FLAGS := 536870912, DN := 1, STATE := 1);
   BAxisSODelay : TIMER := (PRE := 200);
   BAxisStop : MOTION_INSTRUCTION := (FLAGS := 33554432);
   BBayPos : DINT;
   BCompare : REAL;
   BCoordSetup : BOOL;
   BEnableONS : BOOL := 1;
   BEnd : DINT := 6;
   BgridLoc : DINT;
   BInc : DINT;
   BlowerTm : TIMER := (PRE := 300000, ACC := 300001);
   BlowerTmr : TIMER;
   BPitch : REAL;
   BPos : REAL;
   BrakeTmr : TIMER := (PRE := 200);
   BRange : DINT;
   BReq : DINT := 1;
   BReqPos : REAL;
   BStart : REAL;
   CCoordSetup : BOOL;
   CfgEnd : BayPos;
   CfgStrt : BayPos;
   CfgTtlAAxis : DINT := 41;
   CfgTtlBAxis : DINT := 9;
   CFinalPos : DINT := -194536;
   CGridLoc : DINT;
   CHomePos : DINT := 1592;
   CInc : DINT;
   CommandReq : DINT := 4;
   Configuration : Configuration := (MaxASpeed := 75.0, MaxAAcc := 20.0, MaxADec := 20.0, MaxBSpeed := 25.0, MaxBAcc := 15.0, MaxBDec := 15.0);
   CPosHighLim : DINT := -191536;
   CPosLowLim : DINT := -197536;
   CPosSpeed2Tol : DINT := 55000;
   CPosTolerance : DINT := 3000;
   Crane : MOTION_GROUP;
   CReq : DINT;
   CReqPos : DINT := -196128;
   CurrentAPos : DINT := 486;
   CurrentBPos : DINT;
   CurrentCPos : DINT;
   CurrentTask : Task := (Command := 4, BayAPos := 5, BayBPos := 1);
   Demo : BOOL;
   DemoDP : Task[3] := ([0].Command := 1, [0].BayBPos := 3, [0].BayCPos := 1, [1].Command := 2, [1].BayBPos := 1, [1].BayCPos := 1, [2].Command := 4, [2].BayAPos := 10, [2].BayBPos := 3);
   DemoOns : BOOL;
   DemoPU : Task[3] := ([0].Command := 4, [0].BayAPos := 25, [0].BayBPos := 9, [1].Command := 1, [1].BayBPos := 2, [1].BayCPos := 1, [2].Command := 2, [2].BayBPos := 4, [2].BayCPos := 1);
   DepositReq : BOOL;
   DisableAftScanner : BOOL := 1;
   DisableScanners : BOOL;
   DPCntr : DINT := 4;
   DPReg : BOOL;
   DriveEnabled : BOOL;
   DrivesOn : BOOL;
   epc_temp : BOOL := 1;
   EStop : DCI_STOP := (ChannelA := 1, ChannelB := 1, InputStatus := 1, RestartType := 1, ColdStartType := 1, DiscrepancyTime := 30, O1 := 1);
   EStop_SafetyGate : DCI_STOP := (InputStatus := 1, RestartType := 1, ColdStartType := 1, SafetyFunction := 1, DiscrepancyTime := 1000);
   ExtendSpatula : BOOL;
   FootSwitch : ALIAS FOR ShuttleIO:9:I.Pt04Data;
   ForeAreaRst : ALIAS FOR ShuttleIO:8:O.Pt00Data;
   ForeAreaScanner : DCI_STOP := (ChannelA := 1, ChannelB := 1, InputStatus := 1, RestartType := 1, ColdStartType := 1, SafetyFunction := 3, DiscrepancyTime := 500, O1 := 1);
   ForeAreaZn1 : ALIAS FOR ShuttleIO:8:O.Pt02Data;
   ForeAreaZn2 : ALIAS FOR ShuttleIO:10:O.0;
   ForeAreaZn4 : ALIAS FOR ShuttleIO:8:O.Pt03Data;
   FrntAreaWarn : ALIAS FOR ShuttleIO:9:I.Pt00Data;
   FwdEndZn : BOOL;
   FwdEndZone : BOOL;
   GenSafeEn : BOOL;
   GZReset : BOOL;
   GZSafetyReset : BOOL;
   GZSet : BOOL;
   GZSetEnable : BOOL;
   GZSetEnONS : BOOL;
   GZtest : BOOL;
   gztest2 : BOOL := 1;
   GZTest3 : BOOL := 1;
   HighSpdFwd : BOOL;
   HighSpdRev : BOOL;
   HighSpeedFwd : BOOL;
   HighSpeedRev : BOOL;
   HM1734WM1_A : DINT[9] := ([2] := 3, [5] := -1);
   HM1734WM1_B : DINT[2];
   HMI_Commands : HMI_Commands := (GoToALocation := 5, GoToBLocation := 1, XLftStrainScaleSet := 5000, XRtStrainScaleSet := 5000, ZForeRtStrainScaleSet := 5000, ZForeLftStrainScaleSet := 5000, ZAftRtStrainScaleSet := 5000, ZAftLftStrainScaleSet := 5000, XStrainLeftMvV := 1.6333444, XStrainRightMvV := 2.005, ZAftStrainLeftMvV := 2.005, ZAftStrainRightMvV := 2.005, ZForeStrainLeftMvV := 2.005, ZForeStrainRightMvV := 2.005, ManMode := 1, XStRunMode := 1, ZAftStRunMode := 1, ZForStRunMode := 1);
   HMI_Faults : HMI_Faults := (ZAxisDnEOT := 1);
   HMI_Status : HMI_Status := (CurrentAPos := 451.0, CurrentBPos := 21.0, XStrainLeftWeight := 1631, XStrainRightWeight := 1192, ZAftStrainLeftWeight := 1464, ZAftStrainRightWeight := 1205, ZForeStrainLeftWeight := 1320, ZForeStrainRightWeight := 1318, QueuedTasks := 15, CurrentTaskCommand := 4, CurrentTaskBayAPos := 5, Auto := 1, SpatulaHome := 1, FrontAreaWarn := 1, RearAreaWarn := 1);
   HMIData : HMI_Data := (Status.CurrentAPos := 24.549124, Status.CurrentBPos := 0.021048348, Status.XStrainLeftWeight := 1541, Status.XStrainRightWeight := 1413, Status.ZAftStrainLeftWeight := 1467, Status.ZAftStrainRightWeight := 884, Status.ZForeStrainLeftWeight := 795, Status.ZForeStrainRightWeight := 882, Status.AAxisStatus := 9, Status.BAxisStatus := 9, Status.CurrentTaskCommand := 4, Status.CurrentTaskBayAPos := 5, Status.CurrentTaskBayBPos := 1, Status.BackGateInstalled := 1, Status.SpatulaHome := 1, Faults.EstopSafetyGate := 1, Faults.ShuttleFault := 1, Faults.ZAxisDnEOT := 1);
   HMIMsgCtrl : MESSAGE;
        MessageParameters(ServiceCode := 16#004d, LocalElement := HMIData, ...)
   HMITmr : TIMER := (PRE := 500, ACC := 62, EN := 1, TT := 1);
   HomeLowLim : DINT := -2000;
   HomeSpatula : BOOL;
   Horn : ALIAS FOR ShuttleIO:5:O.1;
   Inc : DINT;
   InitialXBrkRls : BOOL;
   InitialZBrkRls : BOOL;
   JogAAxisEn : BOOL;
   JogAcc : DINT;
   JogAct : BOOL;
   JogActive : BOOL;
   JogARev : BOOL := 1;
   JogBAxisEn : BOOL := 1;
   JogBFwd : BOOL := 1;
   JogBRev : BOOL;
   JogConfiguration : Configuration := (MaxASpeed := 15.0, MaxAAcc := 20.0, MaxADec := 40.0, AAccelJerk := 40.0, ADecelJerk := 40.0, MaxBSpeed := 8.0, MaxBAcc := 10.0, MaxBDec := 35.0, BAccelJerk := 60.0, BDecelJerk := 40.0);
   JogDec : DINT;
   JogEnabled : BOOL;
   JogReleaseSBrk : BOOL;
   JogSpeed : DINT;
   Last : DINT := 99;
   LastAAxErr : DINT := 82;
   LastAAxExErr : DINT;
   LastAAxFlt : DINT := 32;
   LastBAxFlt : DINT := 32;
   LastMessageReceiveSequence : DINT := 57738;
   LiftStrainFault : BOOL;
   LiftStrainOK : BOOL := 1;
   LiftStrnOK : BOOL := 1;
   LightCur1 : ALIAS FOR StationaryIO:7:I.Pt06Data;
   LightCur2 : ALIAS FOR StationaryIO:7:I.Pt07Data;
   LightCurEN : ALIAS FOR StationaryIO:6:O.Pt07Data;
   LoadaTask : BOOL;
   LoadTask : Task := (Command := 4, BayAPos := 5, BayBPos := 1);
   LockRelease : ALIAS FOR StationaryIO:7:I.Pt04Data;
   LS_40030 : ALIAS FOR StationaryIO:1:I.0;
   LS_40040 : ALIAS FOR StationaryIO:1:I.1;
   ManConfig : Configuration := (MaxASpeed := 75.0, MaxAAcc := 20.0, MaxADec := 20.0, MaxBSpeed := 25.0, MaxBAcc := 15.0, MaxBDec := 15.0);
   ManGateClosed : ALIAS FOR ShuttleIO:9:I.Pt02Data;
   ManMode : BOOL := 1;
   ManOnBoard : ALIAS FOR ShuttleIO:5:O.5;
   MasterReset : BOOL;
   MatrixSetup : BOOL;
   MaxA : DINT;
   MaxB : DINT;
   MaxC : DINT;
   MechBrkRel : BOOL;
   Messaging : Messaging;
   MoveComplete : BOOL := 1;
   MoveInProcess : BOOL;
   MoveReadly : BOOL := 1;
   MoveReady : BOOL;
   MoveRequested : BOOL;
   MoveSafetyEnable : BOOL;
   MoveToPos : DINT;
   MsgTimer : TIMER := (PRE := 1000);
   MtrEndDsbleZn : REAL;
   NewAPos : DINT := 30;
   NewBPos : DINT := 7;
   NewCmnd : DINT := 4;
   NewCPos : DINT;
   OperatorDN : BOOL;
   Override : BOOL;
   PalmButtonLeft : ALIAS FOR ShuttleIO:9:I.Pt07Data;
   PalmButtonRight : ALIAS FOR ShuttleIO:9:I.Pt06Data;
   PalmButtons : DCI_STOP := (InputStatus := 1, RestartType := 1, ColdStartType := 1, SafetyFunction := 100, DiscrepancyTime := 3000);
   PDSimTmr : TIMER := (PRE := 3000, ACC := 1964, EN := 1, TT := 1);
   PnlEndDsbleZn : REAL := 836.0;
   PorDInProc : BOOL;
   PorDStepTemp : BOOL := 1;
   PorDStop : BOOL;
   PositionFlt : BOOL;
   ProxPwr : ALIAS FOR StationaryIO:6:O.Pt00Data;
   PUCntr : DINT := 5;
   Pulse : TIMER := (PRE := 500, ACC := 3, EN := 1, TT := 1);
   PulseBit : BOOL := 1;
   PUReg : BOOL;
   RearAreaWarn : ALIAS FOR ShuttleIO:9:I.Pt05Data;
   ReceiveMessage : Messaging := (Sequence := 57738);
   ReceiveMessageCommand : MESSAGE;
        MessageParameters(ServiceCode := 16#004c, LocalElement := ReceiveMessage.Command, DestinationTag := ReceiveMessage.Command, ...)
   ReleaseGate : ALIAS FOR StationaryIO:6:O.Pt00Data;
   ReleasePosition : DINT;
   ReleaseSpatBrk : BOOL;
   ResetArea : BOOL;
   ResetSafety : BOOL;
   ResetTmr : TIMER := (PRE := 500);
   RetractSpatula : BOOL;
   Rev : BOOL;
   RowObstruction : BOOL;
   RPE_400140 : ALIAS FOR StationaryIO:2:I.0;
   RPE_400150 : ALIAS FOR StationaryIO:2:I.1;
   RPE_400160 : ALIAS FOR StationaryIO:2:I.2;
   RPE_400170 : ALIAS FOR StationaryIO:2:I.3;
   RPE_400180 : ALIAS FOR StationaryIO:2:I.4;
   RPE_400190 : ALIAS FOR StationaryIO:2:I.5;
   RPE_400200 : ALIAS FOR StationaryIO:2:I.6;
   RPE_400210 : ALIAS FOR StationaryIO:2:I.7;
   RPE_400280 : ALIAS FOR StationaryIO:3:I.0;
   RPE_400290 : ALIAS FOR StationaryIO:3:I.1;
   RPE_400300 : ALIAS FOR StationaryIO:3:I.2;
   RPE_400310 : ALIAS FOR StationaryIO:3:I.3;
   RPE_400320 : ALIAS FOR StationaryIO:3:I.4;
   RPE_400330 : ALIAS FOR StationaryIO:3:I.5;
   RPE_400340 : ALIAS FOR StationaryIO:3:I.6;
   RPE_400350 : ALIAS FOR StationaryIO:3:I.7;
   RPE_400390 : ALIAS FOR StationaryIO:4:I.0;
   RPE_400400 : ALIAS FOR StationaryIO:4:I.1;
   RPE_400410 : ALIAS FOR StationaryIO:4:I.2;
   SafetyGate1 : ALIAS FOR StationaryIO:7:I.Pt00Data;
   SafetyGate2 : ALIAS FOR StationaryIO:7:I.Pt01Data;
   SafetyLaserAft1 : ALIAS FOR ShuttleIO:7:I.Pt04Data;
   SafetyLaserAft2 : ALIAS FOR ShuttleIO:7:I.Pt05Data;
   SafetyLaserFore1 : ALIAS FOR ShuttleIO:7:I.Pt00Data;
   SafetyLaserFore2 : ALIAS FOR ShuttleIO:7:I.Pt01Data;
   SafetyReset : ALIAS FOR StationaryIO:7:I.Pt03Data;
   SafetyResetOns : BOOL := 1;
   SendMessage : Messaging := (Command := 10, CoordinateA := 8, Sequence := 66183562);
   SendMessageCommand : MESSAGE;
        MessageParameters(ServiceCode := 16#004b, LocalElement := SendMessage, DestinationTag := ReceiveMessage, ...)
   SetupEnable : BOOL;
   ShuttleFault : ALIAS FOR ShuttleIO:5:O.3;
   SpatInTmr : TIMER := (PRE := 10000);
   SpatOutTmr : TIMER := (PRE := 10000);
   SpatSimHome : BOOL;
   SpatulaBrake : ALIAS FOR ShuttleIO:5:O.6;
   SpatulaExtendComp : BOOL;
   SpatulaExtended : BOOL;
   SpatulaHome : ALIAS FOR ShuttleIO:2:I.4;
   SpatulaStopped : BOOL;
   Start : ALIAS FOR StationaryIO:7:I.Pt02Data;
   StationaryFault : BOOL := 1;
   StationaryFlt : BOOL := 1;
   StationaryHorn : BOOL;
   StationaryHrn : BOOL;
   StationaryManOn : BOOL;
   StationaryMnOn : BOOL;
   StationaryRn : BOOL;
   StationaryRun : BOOL;
   StationaryWarn : BOOL;
   StationaryWrn : BOOL;
   Stop : ALIAS FOR StationaryIO:7:I.Pt05Data;
   StrainFltTtl : DINT := 4;
   Sts_ASRS_InputsOk : BOOL;
   SUIndPos : BOOL;
   SystemRunning : ALIAS FOR ShuttleIO:5:O.0;
   TaskFIFO : CONTROL := (LEN := 100, EU := 1, EM := 1);
   TaskFile : Task[100];
   TaskInProcess : BOOL := 1;
   temp_DINT1 : DINT := 3;
   temp_DINT2 : DINT := -1;
   temp_DINT3 : DINT := 1;
   temp_DINT4 : DINT := -1;
   temp_Float1 : REAL := inf;
   temp_Float1a : REAL := inf;
   temp_Float2 : REAL := inf;
   temp_Float2a : REAL := inf;
   temp_Float3 : REAL;
   temp_Float3a : REAL;
   test : BOOL;
   test12 : BOOL;
   test2 : BOOL;
   testgz : DINT := 2147483647;
   testgz1 : BOOL := 1;
   TestRun : Task[20] := ([0].Command := 4, [0].BayAPos := 27, [0].BayBPos := 8, [1].Command := 4, [1].BayAPos := 15, [1].BayBPos := 1, [2].Command := 4, [2].BayAPos := 15, [2].BayBPos := 7, [3].Command := 4, [3].BayAPos := 34, [3].BayBPos := 1, [4].Command := 4, [4].BayAPos := 7, [4].BayBPos := 6, [5].Command := 4, [5].BayAPos := 5, [5].BayBPos := 7, [6].Command := 4, [6].BayAPos := 28, [6].BayBPos := 4, [7].Command := 4, [7].BayAPos := 12, [7].BayBPos := 2, [8].Command := 4, [8].BayAPos := 20, [8].BayBPos := 3, [9].Command := 4, [9].BayAPos := 12, [9].BayBPos := 9, [10].Command := 4, [10].BayAPos := 33, [10].BayBPos := 5, [11].Command := 4, [11].BayAPos := 25, [11].BayBPos := 3, [12].Command := 4, [12].BayAPos := 18, [12].BayBPos := 1, [13].Command := 4, [13].BayAPos := 30, [13].BayBPos := 1, [14].Command := 4, [14].BayAPos := 22, [14].BayBPos := 7, [15].Command := 4);
   TestStop : BOOL;
   TestStrain : BOOL;
   testtgl : BOOL;
   TestXBrk : BOOL;
   TestZBrk : BOOL;
   TreadPlate : BOOL;
   TtlCol : DINT;
   TtlRow : DINT;
   UnBindInProc : BOOL;
   UnBindMotnInProc : BOOL := 1;
   Uninhibit : BOOL;
   VFDReset : ALIAS FOR ShuttleIO:6:O.Pt00Data;
   XAccuracy : REAL := 0.25;
   XAxisBrk : ALIAS FOR ShuttleIO:5:O.4;
   XAxisCommands : MESSAGE;
        MessageParameters(ServiceCode := 16#0010, LocalElement := MoveToPos, ...)
   XAxisEOTFault : BOOL;
   XAxisEOTFlt : BOOL;
   XAxisMtrSideEOT : ALIAS FOR ShuttleIO:2:I.6;
   XAxisPnlSideEOT : ALIAS FOR ShuttleIO:2:I.7;
   XAxisSafeStop : CONFIGURABLE_ROUT := (Actuate := 1, Feedback1 := 1, Feedback2 := 1, OutputStatus := 1, FeedbackReactionTime := 500, DiagnosticCode := 32);
   XAxisVFDSS01 : ALIAS FOR ShuttleIO:6:O.Pt04Data;
   XAxisVFDSS02 : ALIAS FOR ShuttleIO:6:O.Pt05Data;
   XBrakeTmr : TIMER := (PRE := 100);
   XHighLimit : REAL := -42.002876;
   XLftCalWeight : DINT;
   XLftRawWeight : DINT;
   XLftTempDint1 : DINT := 25169;
   XLftTempDint2 : DINT := 1541;
   XLftTempFloat1 : REAL := 1.2244815;
   XLftTempFloat2 : REAL := 30818.975;
   XLftTempFloat3 : REAL := 0.05;
   XLowLimit : REAL := -42.502876;
   XLtCTTmr : TIMER := (PRE := 1000);
   XLtTTmr : TIMER := (PRE := 1000);
   XPosHoldTmr : TIMER := (PRE := 20000);
   XRgtTempDint1 : DINT := 28331;
   XRgtTempDint2 : REAL := 1413.0175;
   XRgtTempFloat1 : REAL := 0.9975062;
   XRgtTempFloat2 : REAL := 28260.348;
   XRgtTempFloat3 : REAL := 0.05;
   XRtCalWeight : DINT;
   XRtCTTmr : TIMER := (PRE := 1000);
   XRtRawWeight : DINT;
   XRtTTmr : TIMER := (PRE := 1000);
   XStCalMode : ALIAS FOR StationaryIO:5:O.Data[0].0;
   XStLftSignRun : ALIAS FOR StationaryIO:5:I.Data[7].7;
   XStrain : Strain := (LeftScaleSet := 5000, LeftWeight := 1541, LeftRaw := 25171, LeftCal := -1, RightScaleSet := 5000, RightWeight := 1413, RightRaw := 28331, LeftMvV := 1.6333444, RightMvV := 2.005);
   XStrainHigh : DINT := 2500;
   XStrainLeftMax : DINT := 551017;
   XStrainLeftMin : DINT := 37;
   XStrainLow : DINT := 200;
   XStrainRightMax : DINT := 448878;
   XStrainRightMin : DINT := 2;
   XStRtSignRun : ALIAS FOR StationaryIO:5:I.Data[11].7;
   XStRunMode : ALIAS FOR StationaryIO:5:O.Data[0].1;
   XTensionOK : BOOL := 1;
   ZAccuracy : REAL := 0.25;
   ZADisengage : BOOL;
   ZAftLeftOK : BOOL := 1;
   ZAftLtCTTmr : TIMER := (PRE := 1000);
   ZAftLtTTmr : TIMER := (PRE := 2000);
   ZAftRightOK : BOOL := 1;
   ZAftRtCTTmr : TIMER := (PRE := 1000);
   ZAftRtTTmr : TIMER := (PRE := 1000);
   ZAftStCalMode : ALIAS FOR ShuttleIO:4:O.Data[0].0;
   ZAftStLftSignRun : ALIAS FOR ShuttleIO:4:I.Data[7].7;
   ZAftStrain : Strain := (LeftScaleSet := 5000, LeftWeight := 1466, LeftRaw := 29403, LeftCal := 32, RightScaleSet := 5000, RightWeight := 884, RightRaw := 17724, RightCal := 26, LeftMvV := 2.005, RightMvV := 2.005);
   ZAftStrainLeftMax : DINT := 78202;
   ZAftStrainLeftMin : DINT := 1;
   ZAftStrainRightMax : DINT := 78641;
   ZAftStrainRightMin : DINT := 1;
   ZAftStRtSignRun : ALIAS FOR ShuttleIO:4:I.Data[11].7;
   ZAftStRunMode : ALIAS FOR ShuttleIO:4:O.Data[0].1;
   ZALftTempDint1 : DINT := 29403;
   ZALftTempDint2 : DINT := 1466;
   ZALftTempFloat1 : REAL := 0.9975062;
   ZALftTempFloat2 : REAL := 29329.676;
   ZALftTempFloat3 : REAL := 0.05;
   ZARgtTempDint1 : DINT := 17725;
   ZARgtTempDint2 : DINT := 884;
   ZARgtTempFloat1 : REAL := 0.9975062;
   ZARgtTempFloat2 : REAL := 17680.797;
   ZARgtTempFloat3 : REAL := 0.05;
   ZAxisBrk : ALIAS FOR ShuttleIO:5:O.7;
   ZAxisDnEOT : ALIAS FOR ShuttleIO:1:I.1;
   ZAxisEnabled : BOOL;
   ZAxisEOTFault : BOOL;
   ZAxisEOTFlt : BOOL;
   ZAxisSafetyDisengage : BOOL;
   ZAxisSafetyLatches : ALIAS FOR ShuttleIO:6:O.Pt07Data;
   ZAxisUpEOT : ALIAS FOR ShuttleIO:1:I.0;
   Zero : DINT;
   ZFLftTempDint1 : DINT := 15935;
   ZFLftTempDint2 : DINT := 795;
   ZFLftTempFloat1 : REAL := 0.9975062;
   ZFLftTempFloat2 : REAL := 15895.262;
   ZFLftTempFloat3 : REAL := 0.05;
   ZForeLeftOK : BOOL := 1;
   ZForeRightOK : BOOL := 1;
   ZForeStCalMode : ALIAS FOR ShuttleIO:3:O.Data[0].0;
   ZForeStLftSignRun : ALIAS FOR ShuttleIO:3:I.Data[7].7;
   ZForeStrain : Strain := (LeftScaleSet := 5000, LeftWeight := 795, LeftRaw := 15935, RightScaleSet := 5000, RightWeight := 882, RightRaw := 17694, LeftMvV := 2.005, RightMvV := 2.005);
   ZForeStrainLeftMax : DINT := 78226;
   ZForeStrainLeftMin : DINT := 1;
   ZForeStrainRightMax : DINT := 2099;
   ZForeStrainRightMin : DINT := 1;
   ZForeStRtSignRun : ALIAS FOR ShuttleIO:3:I.Data[11].7;
   ZForeStRunMode : ALIAS FOR ShuttleIO:3:O.Data[0].1;
   ZForLtCTTmr : TIMER := (PRE := 1000);
   ZForLtTTmr : TIMER := (PRE := 1000);
   ZForRtCTTmr : TIMER := (PRE := 1000);
   ZForRtTTmr : TIMER := (PRE := 1000);
   ZFRgtTempDint1 : DINT := 17695;
   ZFRgtTempDint2 : DINT := 883;
   ZFRgtTempFloat1 : REAL := 0.9975062;
   ZFRgtTempFloat2 : REAL := 17650.873;
   ZFRgtTempFloat3 : REAL := 0.05;
   ZHighLimit : REAL := 0.27104342;
   ZLAfltLft : ALIAS FOR StationaryIO:2:I.0;
   ZLAftLft : ALIAS FOR ShuttleIO:2:I.0;
   ZLAftRgt : ALIAS FOR ShuttleIO:2:I.1;
   ZLAutoDly : DINT := 8000;
   ZLBindTmr : TIMER := (PRE := 1000);
   ZLFault : BOOL;
   ZLForeLft : ALIAS FOR ShuttleIO:2:I.3;
   ZLForeRgt : ALIAS FOR ShuttleIO:2:I.2;
   ZLManDly : DINT := 1000;
   ZLockDelay : TIMER := (PRE := 1000, ACC := 1000);
   ZLockMove : MOTION_INSTRUCTION := (FLAGS := 33554432);
   ZLowLimit : REAL := -0.22895658;
   ZLProxOK : BOOL := 1;
   ZLReqPosition : REAL := 39.185207;
   ZLRetryDelay : TIMER := (PRE := 1000);
   ZLsDisengaged : BOOL;
   ZLsProxOK : BOOL := 1;
   ZPosHoldTmr : TIMER := (PRE := 7000);
   ZStrainHigh : DINT := 2500;
   ZStrainLow : DINT := 80;
   ZTest : DINT := 2147483647;
END_VAR
